// TwinCAT 3 PLC project XtsTransport
// Title: XTS Transport
// Author: D.Hauer
// ProjectVersion: 0.0.1
// Description: basic functionblocks for building XTS transport
// ProgramVersion: 3.1.4024.0
// libraries:
//   Tc2_Math, * (Beckhoff Automation GmbH)
//   Tc2_MC2, * (Beckhoff Automation GmbH)
//   Tc2_Standard, * (Beckhoff Automation GmbH)
//   Tc2_System, * (Beckhoff Automation GmbH)
//   Tc2_Utilities, * (Beckhoff Automation GmbH)
//   Tc3_McCollisionAvoidance, * (Beckhoff Automation GmbH)
//   Tc3_McCoordinatedMotion, * (Beckhoff Automation GmbH)
//   Tc3_Module, * (Beckhoff Automation GmbH)
//   Tc3_XTS_Utility, * (Beckhoff Automation GmbH)
//   VisuDialogs, * (System)
// project tree:
//   / GlobalTextList.TcGTLO, MAIN.TcPOU, PlcTask.TcTTO, PROCESS.TcPOU
//   MSG/ fb_LocalTime.TcPOU (not stored), f_MessageSet.TcPOU (not stored), GVL_MSG.TcGVL (not stored), MessageData.TcPOU (not stored), T_MESSAGE_LIST.TcVIS (not stored)
//   MSG/types/ e_Device.TcDUT (not stored), E_MessageType.TcDUT (not stored), E_MESSAGE_STATE.TcDUT (not stored), e_Subdevice.TcDUT (not stored), ST_Message.TcDUT (not stored)
//   PROCESS/ fb_Process.TcPOU, GVL_PROCESS.TcGVL, I_ExternControl_Process.TcIO, PROCESS_CONSTANTS.TcGVL
//   PROCESS/_types/ E_PROCESS_TYPE.TcDUT (not stored)
//   PROCESS/_Visualization/ PROCESS_CONTROL.TcVIS, PROCESS_XTS_TRANSPORT.TcVIS, T_GROUP_VISU.TcVIS, T_PROCESS_VISU.TcVIS, T_XPU_VISU.TcVIS
//   XTS/CaGroup/ FB_CaGroup.TcPOU, I_XtsTransport_CaGroup.TcIO (not stored)
//   XTS/CaGroup/types/ E_CA_GROUP_STATE.TcDUT (not stored), E_GROUP_CHECK.TcDUT (not stored), ST_GROUP_INFO.TcDUT
//   XTS/ GVL_XTS.TcGVL, XTS_Parameter.TcGVL
//   XTS/Mover/ fb_Mover.TcPOU, fb_MoverCtrl.TcPOU (not stored), I_XtsTransport_Mover.TcIO (not stored)
//   XTS/Mover/types/ E_MOVER_CTRL.TcDUT (not stored), E_MOVER_STATE.TcDUT (not stored), ST_GEAR_DATA.TcDUT (not stored), ST_MOVER_CTRL.TcDUT (not stored), ST_MOVER_INFO.TcDUT (not stored), ST_MOVER_STATE.TcDUT (not stored), ST_MOVE_DATA.TcDUT (not stored)
//   XTS/XtsStation/ fb_Station.TcPOU, I_XtsTransport_Station.TcIO (not stored)
//   XTS/XtsStation/_types/ E_STATION_CTRL.TcDUT (not stored), E_STATION_STATE.TcDUT (not stored), fb_Station_LinkedListCtrl.TcPOU (not stored), I_Station_LinkedList.TcIO (not stored), ST_STATION_CTRL.TcDUT (not stored), ST_STATION_LIST_RESULT.TcDUT (not stored), ST_STATION_MOVER_DATA.TcDUT (not stored), ST_STATION_PARAMETER.TcDUT (not stored), ST_STATION_STATE.TcDUT (not stored), T_NEST_OFFSET.TcDUT (not stored)
//   XTS/_types/ f_MoverIdDetectionModeToString.TcPOU, f_MoverPositionAssignementToString.TcPOU, f_XpuOperationModeToString.TcPOU (not stored), E_PROGRESS.TcDUT (not stored), f_GetProgress.TcPOU (not stored), f_GetState.TcPOU (not stored)
//   XTS/_Visualization/ GROUP_VISU.TcVIS, MOVER_VISU.TcVIS (not stored), STATION_VISU.TcVIS, Visualization Manager.TcVMO (not stored), XTS_TRANSPORT.TcVIS (not stored), XPU_VISU.TcVIS (not stored)
//   XTS/_Visualization/textlists/ TL_E_CTRL_MOVER.TcTLO (not stored), TL_E_CTRL_STATION.TcTLO (not stored), TL_E_CTRL_TRANSPORT.TcTLO (not stored), TL_E_CTRL_XPU.TcTLO (not stored)
//   XTS/Xpu/ fb_Xpu.TcPOU (not stored), fb_XpuCtrl.TcPOU (not stored)
//   XTS/Xpu/types/ E_XPU_CHECK.TcDUT (not stored), E_XPU_CTRL.TcDUT (not stored), E_XPU_INIT.TcDUT (not stored), E_XPU_STATE.TcDUT (not stored), ST_XPU_CTRL.TcDUT (not stored), ST_XPU_INFO.TcDUT (not stored), ST_XPU_STATE.TcDUT (not stored)
//   XTS/XtsTransportUnit/ fb_TransportUnit.TcPOU
//   XTS/XtsTransportUnit/types/ E_XTS_TRANSPORT_CHECK.TcDUT (not stored), E_XTS_TRANSPORT_CTRL.TcDUT (not stored), E_XTS_TRANSPORT_STATE.TcDUT (not stored), ST_XTS_TRANSPORT_CTRL.TcDUT (not stored), ST_XTS_TRANSPORT_STATE.TcDUT (not stored)

CONFIGURATION XtsTransport
    RESOURCE PLC ON TwinCAT3
        TASK PlcTask(INTERVAL := T#2ms, PRIORITY := 15);
        PROGRAM MAIN WITH PlcTask : MAIN;
        PROGRAM PROCESS WITH PlcTask : PROCESS;
    END_RESOURCE
END_CONFIGURATION

// ---- XTS/CaGroup/types/ST_GROUP_INFO.TcDUT
TYPE ST_GROUP_INFO :
STRUCT
  GroupStatusValid,
  GroupStatusBusy,
  GroupMoving, 
  GroupHoming, 
  GroupErrorStop, 
  GroupNotReady, 
  GroupStandby, 
  GroupStopping,
 
  GroupDisabled, 
  AllAxesStanding, 
  ConstantVelocity, 
  Accelerating, 
  Decelerating, 
  InPosition, 
  GroupError					  : BIT; 

  GroupErrorId					: UDINT;

  AxisCount      				: UDINT;
  AxisCountEnabled      : UDINT;

  {attribute 'displaymode':='hex'}
  CaGroupOID            : OTCID;

  CaGroupState          : E_CA_GROUP_STATE;
END_STRUCT
END_TYPE

// ---- PROCESS/GVL_PROCESS.TcGVL
{attribute 'qualified_only'}
VAR_GLOBAL

  Process           : ARRAY[1..MAX_PROCESS] OF fb_Process;  // handshake multiple XTS stations (ST_STATION_CTRL / ST_STATION_STATE)
  ItfProcess        : ARRAY[1..MAX_PROCESS] OF I_ExternControl_Process;

  StationsEnabled   : ARRAY[1..MAX_STATION] OF BOOL;        // read only; every process writes internally onto here the bits in MAIN.wEnableProcess
  MoverPerMinute    : ARRAY[1..MAX_STATION] OF UINT;
END_VAR

// ---- PROCESS/PROCESS_CONSTANTS.TcGVL
//{attribute 'qualified_only'}
VAR_GLOBAL CONSTANT
  MAX_PROCESS       : UINT := 12;

END_VAR

// ---- XTS/GVL_XTS.TcGVL
{attribute 'qualified_only'}
VAR_GLOBAL
  //---------------------------------------------------------------------------
  // XTS Station
  //  - handshakes mover in station with extern control
  //  - station parameters (positions, gap, dyn. constraints, description...)
  StationStart        : ST_STATION_PARAMETER;   // Xts transport is sending all mover to this position (CMD_TRANSPORT_START)

  // station handshaking with mover and extern process
  // station sends mover to target station/WaitPos
  // station adds mover data to LinkedList.AddTail() of target station
  Station             : ARRAY[1..MAX_STATION] OF fb_Station;
  StationList         : ARRAY[1..MAX_STATION] OF fb_Station_LinkedListCtrl;

  StationQueue        : ARRAY[1..MAX_STATION]    OF 
                        ARRAY[1..MAX_LIST_NODES] OF ST_STATION_MOVER_DATA;

  // interface for access to List methods
  StationListItf      : ARRAY[1..MAX_STATION] OF I_Station_LinkedList;

  // interface for access to station methods
  StationCtrlItf      : ARRAY[1..MAX_STATION] OF I_XtsTransport_Station;

  // ctrl / state datafields for extern control
  StationCtrl         : ARRAY[1..MAX_STATION] OF ST_STATION_CTRL;   // control for extern to write
  StationState        : ARRAY[1..MAX_STATION] OF ST_STATION_STATE;  // state for extern to read

  // station parameter
  StationParameter    : ARRAY[1..MAX_STATION] OF ST_STATION_PARAMETER;

  // static position offsets in stations
  PositionOffset      : ARRAY[1..MAX_STATION] OF T_NEST_OFFSET;


  //---------------------------------------------------------------------------
  // XTS
  // XTS TransportUnit
  //  - handles request for XPU, Group, Mover, StartUp, ReStart
  XtsTransport        : fb_TransportUnit;         // manages members of XTS transport for extern to access

  XtsTransportCtrl    : ST_XTS_TRANSPORT_CTRL;    // control of XTS transport for extern to write
  XtsTransportState   : ST_XTS_TRANSPORT_STATE;   // state   of XTS transport for extern to read


  //---------------------------------------------------------------------------
  // XPU
  // XTS-Utility checks
  Xpu             : fb_XpuCtrl;

  XpuCtrl         : ST_XPU_CTRL;
  XpuState        : ST_XPU_STATE;
  XpuInfo         : ST_XPU_INFO;
  XpuModules      : ARRAY[1..MAX_MODULE] OF Tc3_XTS_Utility.ST_InfoDataView;


  //---------------------------------------------------------------------------
  // Collision avoidance group CA
  //
  // - add mover to group
  // - build group
  // - clear group
  CaGroup         : FB_CaGroup;                   // cyclic check of CaGroup state and errors; carries methods for handling CaGroup
  CaGroupItf      : I_XtsTransport_CaGroup;       // Interface used by fb_TransportUnit

  // cyclic mapping to MOTION/Objects/CaGroup 
  CaGroupRef      : Tc3_McCoordinatedMotion.AXES_GROUP_REF;

  // Info data from CaGroup FB
  CaGroupInfo     : ST_GROUP_INFO;                // cyclic info about CaGroup for fb_TransportUnit to read
  //---------------------------------------------------------------------------

  //---------------------------------------------------------------------------
  // MC2 encapsulation, CA movement
  Mover           : ARRAY[1..MAX_MOVER] OF fb_MoverCtrl;    // MC and CA methods for mover; cyclic check for individual command on mover

  MoverCtrl       : ARRAY[1..MAX_MOVER] OF ST_MOVER_CTRL;   // control of individual mover for extern to write
  MoverState      : ARRAY[1..MAX_MOVER] OF ST_MOVER_STATE;  // state   of individual mover for extern to read

  MoverItf        : ARRAY[1..MAX_MOVER] OF I_XtsTransport_Mover;  // Interface used by fb_TransportUnit

  LastPosition    : ARRAY[1..MAX_MOVER] OF LREAL;           // on execute of any movement, value is saved here (used by fb_Mover)
  LastGap         : ARRAY[1..MAX_MOVER] OF LREAL;           // on execute of any movement, value is saved here (used by fb_Mover)

  MoverInfo       : ARRAY[1..MAX_MOVER] OF ST_MOVER_INFO;   // cyclic info about mover for extern to read

  MoveData        : ARRAY[1..MAX_MOVER] OF ST_MOVE_DATA;    // dynamic constraints for move commands
  GearData        : ARRAY[1..MAX_MOVER] OF ST_GEAR_DATA;    // dynamic constraints and positions for GearIn/GearInPosCa
  
  // cyclic mapping to MOTION/Axes
  AxisRefMover    : ARRAY[1..MAX_MOVER] OF Tc2_MC2.AXIS_REF;
  //---------------------------------------------------------------------------
END_VAR

// ---- XTS/XTS_Parameter.TcGVL
//{attribute 'qualified_only'}
VAR_GLOBAL CONSTANT
// HAUD 2024 08 09
//
//    XTS_TRANSPORT_LAYER project
//    
//    MIT License
//    
//    Copyright (c) 2024 HAUD
//    
//    Permission is hereby granted, free of charge, to any person obtaining a copy
//    of this software and associated documentation files (the "Software"), to deal
//    in the Software without restriction, including without limitation the rights
//    to use, copy, modify, merge, publish, distribute, sublicense, and/or sell
//    copies of the Software, and to permit persons to whom the Software is
//    furnished to do so, subject to the following conditions:
//    
//    The above copyright notice and this permission notice shall be included in all
//    copies or substantial portions of the Software.
//    
//    THE SOFTWARE IS PROVIDED "AS IS", WITHOUT WARRANTY OF ANY KIND, EXPRESS OR
//    IMPLIED, INCLUDING BUT NOT LIMITED TO THE WARRANTIES OF MERCHANTABILITY,
//    FITNESS FOR A PARTICULAR PURPOSE AND NONINFRINGEMENT. IN NO EVENT SHALL THE
//    AUTHORS OR COPYRIGHT HOLDERS BE LIABLE FOR ANY CLAIM, DAMAGES OR OTHER
//    LIABILITY, WHETHER IN AN ACTION OF CONTRACT, TORT OR OTHERWISE, ARISING FROM,
//    OUT OF OR IN CONNECTION WITH THE SOFTWARE OR THE USE OR OTHER DEALINGS IN THE
//    SOFTWARE.

  Version             : STRING  := '4.0.1';

  MAX_MOVER           : UINT    := TO_UINT(Tc3_XTS_Utility.TcIoXtsEnvironmentParameterList.MaxXtsMoversPerXpu);
  MAX_MODULE          : UINT    := TO_UINT(Tc3_XTS_Utility.TcIoXtsEnvironmentParameterList.MaxModulesPerPart);
  MAX_PART            : UINT    := TO_UINT(Tc3_XTS_Utility.TcIoXtsEnvironmentParameterList.MaxXtsPartsPerXpu);
  MAX_TRACK           : UINT    := TO_UINT(Tc3_XTS_Utility.TcIoXtsEnvironmentParameterList.MaxXtsTracksPerXpu);
  MAX_GROUP           : UINT    := TO_UINT(Tc3_XTS_Utility.TcIoXtsEnvironmentParameterList.MaxXtsCaGroup);

  MAX_INFO_SERVER     : UINT    := TO_UINT(Tc3_XTS_Utility.TcIoXtsEnvironmentParameterList.MaxXtsInfoServer);
  MAX_INFO_STATION    : UINT    := TO_UINT(Tc3_XTS_Utility.TcIoXtsEnvironmentParameterList.MaxXtsInfoStation);
  MAX_INFO_STOP_POS   : UINT    := TO_UINT(Tc3_XTS_Utility.TcIoXtsEnvironmentParameterList.MaxXtsStopPositionsPerStation);


  MAX_STATION         : UINT    := 28;
  MAX_STATION_NEST    : UINT    := TO_UINT(SIZEOF(ST_STATION_STATE.nMask)*8);
  // MAX_LIST_NODES      : UINT    := MAX_MOVER;
  MAX_LIST_NODES      : UINT    := 50; // visualization can not handle access to MAX_MOVER
  MAX_MASTER          : UINT    := 1;
END_VAR

// ---- PROCESS/I_ExternControl_Process.TcIO
INTERFACE I_ExternControl_Process

METHOD PUBLIC DelBitDWord : DWORD
VAR_INPUT
  inVal   : DWORD;
  bitNo   : DWORD;
END_VAR
END_METHOD

PROPERTY EnableProcess : dword
GET
END_GET
SET
END_SET
END_PROPERTY

METHOD PUBLIC GetBitDWord : BOOL
VAR_INPUT
  inVal   : DWORD;
  bitNo   : DINT;
END_VAR
END_METHOD

METHOD PUBLIC Init : BOOL
END_METHOD

PROPERTY MoverCountInQueue : uint
GET
END_GET
END_PROPERTY

PROPERTY MoverInQueue : Bool
GET
END_GET
END_PROPERTY

PROPERTY ProcessCmd : E_STATION_CTRL
SET
END_SET
END_PROPERTY

PROPERTY ProcessPerMinute : uint
GET
END_GET
END_PROPERTY

PROPERTY ProcessState : E_STATION_STATE
GET
END_GET
END_PROPERTY

PROPERTY ProcessType : e_process_type
GET
END_GET
SET
END_SET
END_PROPERTY

METHOD PUBLIC SetBitDWord : DWORD
VAR_INPUT
  inVal   : DWORD;
  bitNo   : DWORD;
END_VAR
END_METHOD

METHOD PUBLIC SetBitWord : WORD
VAR_INPUT
  inVal   : WORD;
  bitNo   : DINT;
END_VAR
END_METHOD

PROPERTY StationCount : uint
GET
END_GET
END_PROPERTY

PROPERTY StationFirst : uint
GET
END_GET
SET
END_SET
END_PROPERTY

PROPERTY TargetMask : dword
GET
END_GET
SET
END_SET
END_PROPERTY

END_INTERFACE

// ---- MAIN.TcPOU
//---------------------------------------------------------------------------------------------------------------
//
//  HAUD 2024.03.18
//
//  - XTS_TRANSPORT_LAYER
//  - transport layer members:
//    - CaGroup
//      - access to Group functions
//
//    - Mover
//      - access to MC and CA motion functions
//
//    - Xpu (ProcessingUnit)
//      - access to TcCOM Objects in Environment
//
//    - Transport Control Unit
//      - coordinates members to get XTS in defined states
//
//    - Xts Stations
//      - handshakes with extern control for mover transport
//
//  - global datafields for mrmbers in GVL_XTS namespace
//  - global interface datafields for use in members
//  - structures are assigned by reference for every member
//
//---------------------------------------------------------------------------------------------------------------
// HAUD 2024 05 29
//
//    XTS_TRANSPORT_LAYER project
//    
//    MIT License
//    
//    Copyright (c) 2024 HAUD
//    
//    Permission is hereby granted, free of charge, to any person obtaining a copy
//    of this software and associated documentation files (the "Software"), to deal
//    in the Software without restriction, including without limitation the rights
//    to use, copy, modify, merge, publish, distribute, sublicense, and/or sell
//    copies of the Software, and to permit persons to whom the Software is
//    furnished to do so, subject to the following conditions:
//    
//    The above copyright notice and this permission notice shall be included in all
//    copies or substantial portions of the Software.
//    
//    THE SOFTWARE IS PROVIDED "AS IS", WITHOUT WARRANTY OF ANY KIND, EXPRESS OR
//    IMPLIED, INCLUDING BUT NOT LIMITED TO THE WARRANTIES OF MERCHANTABILITY,
//    FITNESS FOR A PARTICULAR PURPOSE AND NONINFRINGEMENT. IN NO EVENT SHALL THE
//    AUTHORS OR COPYRIGHT HOLDERS BE LIABLE FOR ANY CLAIM, DAMAGES OR OTHER
//    LIABILITY, WHETHER IN AN ACTION OF CONTRACT, TORT OR OTHERWISE, ARISING FROM,
//    OUT OF OR IN CONNECTION WITH THE SOFTWARE OR THE USE OR OTHER DEALINGS IN THE
//    SOFTWARE.
//---------------------------------------------------------------------------------------------------------------
PROGRAM MAIN
VAR
	bInit 				: BOOL;
  eInit         : E_PROGRESS;

  nStation,
	nMover,
  nMoverSelected,
  nStationSelected,
  nStationParameter   : UINT;

  sStationText        : STRING(30);

  eTransportState     : E_XTS_TRANSPORT_STATE;
  eTransportResult    : E_PROGRESS;

  eXpuState           : E_XPU_STATE;
  eXpuResult          : E_PROGRESS;
  eXpuCheck           : E_XPU_CHECK;

  eMoverState         : E_MOVER_STATE;
  eMoverResult        : E_PROGRESS;

  sCaGroupState,
  sTransportState,
  sTransportCheck,
  sTransportResult,
  sXpuState,
  sXpuResult,
  sXpuCheck,
  sXpuOpMode,
  sXpuMoverdetectionMode,
  sXpuMoverAssignement,
  sMoverState,
  sMoverResult,
  sStationState,
  sStationStateMask,
  sStationCtrlMask        : STRING;

  bStationEnable,
  bStationEnter,
  bStationStart,
  bStationDone,
  bStationOut,
  bStationGone            : BOOL;

  tStationSelectedQueue   : ARRAY[1..MAX_LIST_NODES] OF ST_STATION_MOVER_DATA;

  tonWriteLog             : Tc2_Standard.TON;
  tWriteLog               : TIME := T#5S;
END_VAR

//############################################################################
// Local time; used for timestamps
//############################################################################
GVL_MSG.fbLocalTime(
                    sLocalTime                => GVL_MSG.sLocalTime, 
                    dtLocalTime               => GVL_MSG.dtLocalTime);
//############################################################################

//############################################################################
// 	example for init sequence
//############################################################################	
IF NOT bInit
THEN
  CASE eInit
  OF
    E_PROGRESS.PROGRESS_INVALID,
    E_PROGRESS.PROGRESS_DONE:         // clear command interface
      eInit                                   := E_PROGRESS.PROGRESS_BUSY;
      GVL_XTS.XpuCtrl.Cmd                     := E_XPU_CTRL.XTS_CMD_NULL;
      GVL_MSG.MessageLevelXpu                 := GVL_MSG.MessageLevel;
      FOR nStation := 1 TO MAX_STATION
      DO
        GVL_MSG.MessageLevelStations[nStation]:= GVL_MSG.MessageLevel;
      END_FOR
      FOR nMover := 1 TO MAX_MOVER
      DO
        GVL_MSG.MessageLevelMovers[nMover]    := GVL_MSG.MessageLevel;
      END_FOR


    E_PROGRESS.PROGRESS_BUSY:         // init Xpu, ProcessingUnit, MotorModules
      eInit                                   := E_PROGRESS.PROGRESS_PREPARE;
      GVL_XTS.XpuCtrl.Cmd                     := E_XPU_CTRL.XTS_CMD_INIT;

    E_PROGRESS.PROGRESS_PREPARE:      // wait for init to be done
      IF (GVL_XTS.XpuState.State      = E_XPU_STATE.XTS_INIT + E_PROGRESS.PROGRESS_DONE)
      THEN
        eInit                                 := E_PROGRESS.PROGRESS_STARTUP;
        GVL_XTS.XpuCtrl.Cmd                   := E_XPU_CTRL.XTS_IDLE;
      END_IF

    E_PROGRESS.PROGRESS_STARTUP:      // assign mover interfaces
      eInit                                   := E_PROGRESS.PROGRESS_CHECK;
      FOR nMover := 1 TO MAX_MOVER
      DO
        GVL_XTS.MoverItf[nMover]              := GVL_XTS.Mover[nMover];
      END_FOR

    E_PROGRESS.PROGRESS_CHECK:        // assign CaGroup interface
      eInit                                   := E_PROGRESS.PROGRESS_OCCUPIED;
      GVL_XTS.CaGroupItf                      := GVL_XTS.CaGroup;

    E_PROGRESS.PROGRESS_OCCUPIED:     // StartStation for XtsTransportCtrl.Cmd := E_XTS_TRANSPORT_CTRL.CMD_TRANSPORT_START;
      eInit                                   := E_PROGRESS.PROGRESS_WORKING;
      // where to start?
      GVL_XTS.XtsTransport.StartStationIndex  := 28;

      // Start Position parameters
      GVL_XTS.StationStart.rPosWait           := GVL_XTS.StationParameter[28].rPosWait;
      GVL_XTS.StationStart.rGap               :=    100.0;
      GVL_XTS.StationStart.rVelo              :=   1250.0;
      GVL_XTS.StationStart.rAccDec            :=  12000.0;
      GVL_XTS.StationStart.rJerk              := 400000.0;

    E_PROGRESS.PROGRESS_WORKING:
      bInit                                           := TRUE;
      eInit                                           := E_PROGRESS.PROGRESS_DONE;
  END_CASE
END_IF

//############################################################################
// 	XTS Transport Unit
//############################################################################
//  - main control function block for transport layer
//  - requires access to member controls
//    - Xpu
//    - CaGroup
//    - Mover
//    - Station Control
//    - Station LinkedList Interface
//############################################################################
//
// cyclic call
GVL_XTS.XtsTransport();

// main control
GVL_XTS.XtsTransport.Ctrl               REF= GVL_XTS.XtsTransportCtrl;   // main control
GVL_XTS.XtsTransport.State              REF= GVL_XTS.XtsTransportState;  // main state
                                        
// member controls                      
GVL_XTS.XtsTransport.XpuCtrl            REF= GVL_XTS.XpuCtrl;
GVL_XTS.XtsTransport.XpuState           REF= GVL_XTS.XpuState;
GVL_XTS.XtsTransport.XpuInfo            REF= GVL_XTS.XpuInfo;
                                        
GVL_XTS.XtsTransport.GroupItf           :=   GVL_XTS.CaGroupItf;
GVL_XTS.XtsTransport.GroupInfo          REF= GVL_XTS.CaGroupInfo;
                                        
GVL_XTS.XtsTransport.MoverItf           REF= GVL_XTS.MoverItf;
GVL_XTS.XtsTransport.MoverInfo          REF= GVL_XTS.MoverInfo;
                                        
GVL_XTS.XtsTransport.StationStart       REF= GVL_XTS.StationStart;      // start position for E_XTS_TRANSPORT_CTRL.CMD_TRANSPORT_START
GVL_XTS.XtsTransport.StationCtrlItf     REF= GVL_XTS.StationCtrlItf;    // station interfaces are required for accessing station methods
GVL_XTS.XtsTransport.StationListsItf    REF= GVL_XTS.StationListItf;    // list interface is required for access to linked list methods
//############################################################################



//############################################################################
// 	XTS Stations
//############################################################################	
FOR nStation := 1 TO MAX_STATION
DO
  GVL_XTS.Station[nStation].StationId   := nStation;
  GVL_XTS.Station[nStation].MessageLevel:= GVL_MSG.MessageLevelStations[nStation];

  GVL_XTS.StationListItf[nStation]      := GVL_XTS.StationList[nStation];   // interfaces for list methods
  GVL_XTS.StationCtrlItf[nStation]      := GVL_XTS.Station[nStation];       // interfaces for station methods

  GVL_XTS.Station[nStation].Ctrl        REF= GVL_XTS.StationCtrl;           // station ctrl from extern
  GVL_XTS.Station[nStation].State       REF= GVL_XTS.StationState;          // station state to extern

  GVL_XTS.Station[nStation].ItfStations REF= GVL_XTS.StationListItf;        // give every station all list interfaces for writing mover tickets
  GVL_XTS.Station[nStation].ItfMover    REF= GVL_XTS.MoverItf;              // give every station all mover interfaces for movement in / out of station
  GVL_XTS.Station[nStation].Mover       REF= GVL_XTS.AxisRefMover;          // AXIS_REF to read infos from
  GVL_XTS.Station[nStation].MoverOffset REF= GVL_XTS.PositionOffset;        // static offsets for all stations, all movers, all stop positions


  GVL_XTS.Station[nStation].StationParameter  REF= GVL_XTS.StationParameter;// give every station all station parameters for sending to WaitPos of target station

  // cyclic call
  GVL_XTS.Station[nStation].Cycle();                                        // cycle for handshaking with extern

  // Queue data for each station
  GVL_XTS.StationQueue[nStation]        := GVL_XTS.StationListItf[nStation].Data;
END_FOR
//############################################################################



//############################################################################
// 	XPU environment
//############################################################################	
GVL_XTS.Xpu.XpuInstance               :=   1;
GVL_XTS.Xpu.MessageLevel              :=   GVL_MSG.MessageLevelXpu;

GVL_XTS.Xpu.Ctrl                      REF= GVL_XTS.XpuCtrl;
GVL_XTS.Xpu.State                     REF= GVL_XTS.XpuState;
GVL_XTS.Xpu.XpuModuleInfoData         REF= GVL_XTS.XpuModules;

GVL_XTS.Xpu.CaGroupOID                :=   GVL_XTS.CaGroup.GroupInfo.CaGroupOID;

// cyclic call
GVL_XTS.Xpu();
GVL_XTS.XpuInfo                       :=   GVL_XTS.Xpu.XpuInfo;
//############################################################################


//############################################################################	
// 	CA-Group Class
//############################################################################	
// assignment
GVL_XTS.CaGroup.AxisRef               REF= GVL_XTS.AxisRefMover;
GVL_XTS.CaGroup.GroupRef              REF= GVL_XTS.CaGroupRef;

GVL_XTS.CaGroup.MessageLevel          :=   GVL_MSG.MessageLevel;

// cyclic call
GVL_XTS.CaGroup.InfoCycle(TRUE); // read group status

// InfoData from group
GVL_XTS.CaGroupInfo                   :=   GVL_XTS.CaGroup.GroupInfo;

// Interface of CaGroup
GVL_XTS.CaGroupItf                    :=   GVL_XTS.CaGroup;
//############################################################################


//############################################################################
// Mover Class	
//############################################################################	
FOR nMover := 1 TO MAX_MOVER
DO
  GVL_XTS.Mover[nMover].MoverId       :=   nMover;
  GVL_XTS.Mover[nMover].RailLength    :=   GVL_XTS.Xpu.RailLength;  // mover needs RailLength, in order to calc absolute position from modulo input
  GVL_XTS.Mover[nMover].MessageLevel  :=   GVL_MSG.MessageLevelMovers[nMover];

  GVL_XTS.Mover[nMover].Ctrl          REF= GVL_XTS.MoverCtrl;       // mover control from extern
  GVL_XTS.Mover[nMover].State         REF= GVL_XTS.MoverState;      // mover state to extern

  GVL_XTS.Mover[nMover].MoveData      REF= GVL_XTS.MoveData;        // dyn constraints for extern to write
  GVL_XTS.Mover[nMover].GearData      REF= GVL_XTS.GearData;        // GearIn/GearInPosCa data fro extern to write

  // assignment	
  GVL_XTS.Mover[nMover].Mover         REF= GVL_XTS.AxisRefMover[nMover];  // axis reference to Mover function block
  GVL_XTS.Mover[nMover].LastGap       REF= GVL_XTS.LastGap[nMover];       // reference to last used gap value datafield
  GVL_XTS.Mover[nMover].LastPosition  REF= GVL_XTS.LastPosition[nMover];  // reference to last position datafield

  GVL_XTS.Mover[nMover].MoverInfo		  REF= GVL_XTS.MoverInfo[nMover];     // refernence to mover info data (ActPos, SetPos, ...)

  GVL_XTS.MoverItf[nMover]            :=   GVL_XTS.Mover[nMover];

  // cyclic call
  GVL_XTS.Mover[nMover].Cycle();  // call AXIS_REF()
  GVL_XTS.Mover[nMover]();        // call Ctrl/State
END_FOR


//############################################################################


//############################################################################
// /logging
//############################################################################
tonWriteLog(IN:= TRUE, PT := tWriteLog);

IF (tonWriteLog.Q)
THEN
  MessageData.bWriteFile      := TRUE;
  tonWriteLog(IN:= FALSE);
END_IF

//-----------------------------------------------------------------------------------------------------------------
// write message list to file
//-----------------------------------------------------------------------------------------------------------------
MessageData(pList			        := ADR(GVL_MSG.Messages),
			      pLocalTime        := ADR(GVL_MSG.dtLocalTime), 
			      bBusy=> );

// clear write trigger
IF MessageData.bWriteFile AND
   MessageData.bDone
THEN
  MessageData.bWriteFile      := FALSE;
END_IF
//############################################################################
// logging/
//############################################################################



//############################################################################
// Visualization data	
//############################################################################	
// get enumerations from XPU for visu:
eTransportState                       := f_GetState   (GVL_XTS.XtsTransportState.State);
eTransportResult                      := f_GetProgress(GVL_XTS.XtsTransportState.State);

eXpuState                             := f_GetState   (GVL_XTS.XpuState.State);
eXpuResult                            := f_GetProgress(GVL_XTS.XpuState.State);

eXpuCheck                             := GVL_XTS.XpuState.Check;

// display xpu state and result in visu
// get strings and info
sCaGroupState                         := TO_STRING(GVL_XTS.CaGroupInfo.CaGroupState);

sTransportState                       := TO_STRING(eTransportState);
sTransportCheck                       := TO_STRING(GVL_XTS.XtsTransportState.Check);
sTransportResult                      := TO_STRING(eTransportResult);

sXpuState                             := TO_STRING(eXpuState);
sXpuResult                            := TO_STRING(eXpuResult);
sXpuCheck                             := TO_STRING(eXpuCheck);

sXpuOpMode                            := GVL_XTS.Xpu.OpModeToString();
sXpuMoverdetectionMode                := GVL_XTS.Xpu.IdDetectionModeToString();
sXpuMoverAssignement                  := GVL_XTS.Xpu.MoverPositionAssignementToString();

nMoverSelected                        := SEL((nMoverSelected<1), nMoverSelected, 1);
nMoverSelected                        := SEL((nMoverSelected>MAX_MOVER), nMoverSelected, MAX_MOVER);

nStationSelected                      := SEL((nStationSelected<1), nStationSelected, 1);
nStationSelected                      := SEL((nStationSelected>MAX_STATION), nStationSelected, MAX_STATION);

bStationEnable                        := SEL((GVL_XTS.StationCtrl[nStationSelected].eCmd = E_STATION_CTRL.STATION_ENABLE),        FALSE, TRUE);
bStationEnter                         := SEL((GVL_XTS.StationCtrl[nStationSelected].eCmd = E_STATION_CTRL.STATION_MOVER_ENTER),   FALSE, TRUE);
bStationStart                         := SEL((GVL_XTS.StationCtrl[nStationSelected].eCmd = E_STATION_CTRL.STATION_PROCESS_START), FALSE, TRUE);
bStationDone                          := SEL((GVL_XTS.StationCtrl[nStationSelected].eCmd = E_STATION_CTRL.STATION_PROCESS_DONE),  FALSE, TRUE);
bStationOut                           := SEL((GVL_XTS.StationCtrl[nStationSelected].eCmd = E_STATION_CTRL.STATION_MOVER_OUT),     FALSE, TRUE);
bStationGone                          := SEL((GVL_XTS.StationCtrl[nStationSelected].eCmd = E_STATION_CTRL.STATION_MOVER_GONE),    FALSE, TRUE);

eMoverState                           := f_GetState   (GVL_XTS.MoverState[nMoverSelected].State);
eMoverResult                          := f_GetProgress(GVL_XTS.MoverState[nMoverSelected].State);

sMoverState                           := TO_STRING(eMoverState);
sMoverResult                          := TO_STRING(eMoverResult);

sStationState                         := TO_STRING(GVL_XTS.StationState[nStationSelected].eState);
sStationStateMask                     := Tc2_Utilities.BYTE_TO_BINSTR(GVL_XTS.StationState[nStationSelected].nMask, 8);
sStationCtrlMask                      := Tc2_Utilities.BYTE_TO_BINSTR(GVL_XTS.StationCtrl[nStationSelected].nMask, 8);

tStationSelectedQueue                 := GVL_XTS.StationQueue[nStationSelected];

END_PROGRAM

// ---- PROCESS.TcPOU
//---------------------------------------------------------------------------------------------------------------
//
//  HAUD 2024.04.13
//
//  - ExternControl for XtsTransport
//
//  - example project for controlling XTS transport layer
//  - transport layer members:
//
//      HAUD 2024 04 30 - introduction of fb_UnitControl as interface to APPLICATION
//
//    - fb_UnitControl
//      - groups commands into sequences for APPLICATION
//      - handles XtsTransport
//      - handles fb_Process
//
//    - fb_Process
//      - groups XtsStations for processes
//      - synced handshakes with all assigned XtsStations
//
//    - Transport Control Unit
//      - mapped from XtsTransport GVL_XTS.TransportCtrl / GVL_XTS.TransportState
//        - Info for CaGroup
//        - Info for Xpu
//
//      - coordinates members to get XTS in defined states
//
//    - Xts Stations
//      - handshakes for mover transport
//
//---------------------------------------------------------------------------------------------------------------
// This SOFTWARE is provided as an Exemple by THE PROVIDER "as is" and "with all faults." THE PROVIDER makes no 
// representations or warranties of any kind concerning the safety, suitability, lack of viruses, inaccuracies, 
// typographical errors, or other harmful components of this SOFTWARE. There are inherent dangers in the use of 
// any software, and you are solely responsible for determining whether this SOFTWARE is compatible with your 
// equipment and other software installed on your equipment. You are also solely responsible for the protection 
// of your equipment and backup of your data, and THE PROVIDER will not be liable for any damages you may suffer 
// in connection with using, modifying, or distributing this SOFTWARE.
//---------------------------------------------------------------------------------------------------------------
PROGRAM PROCESS
VAR
  bInit,
  bStart              : BOOL;       // start bit for AUTO
  eInit               : E_PROGRESS; // process initialization

  eTransportCmd,
  eTransportCmdOld    : E_XTS_TRANSPORT_CTRL; // ctrl input sequence

  eTransportState,
  eTransportStateOld  : E_XTS_TRANSPORT_STATE;// state output sequence

  eTransportResult,
  eStateStart         : E_PROGRESS;

  nProcess,
  nStation            : UINT;

  tProcess            : ARRAY[1..MAX_PROCESS] OF TIME;
  tonProcess          : ARRAY[1..MAX_PROCESS] OF Tc2_Standard.TON;

  {attribute 'displaymode':='bin'}
  wEnableProcess      : ARRAY[1..MAX_PROCESS] OF DWORD;  // switch XTS stations on/off here (one word per process --> max. 16 stations each)

  {attribute 'displaymode':='bin'}
  wInitProcess        : WORD;  // processes init

//  eProcessCmd         : ARRAY[1..MAX_PROCESS] OF E_STATION_CTRL;
//  eProcessState       : ARRAY[1..MAX_PROCESS] OF E_STATION_STATE;

  // visualization vars
  nMoverSelected,
  nStationSelected,
  nProcessSelected,
  nStationParameter,
  nProcessParameter   : UINT;

  eXpuState           : E_XPU_STATE;
  eXpuResult          : E_PROGRESS;
  eXpuCheck           : E_XPU_CHECK;

  eMoverState         : E_MOVER_STATE;
  eMoverResult        : E_PROGRESS;

  sCaGroupState,
  sTransportState,
  sTransportCheck,
  sTransportResult,
  sXpuState,
  sXpuResult,
  sXpuCheck,
  sXpuOpMode,
  sXpuMoverdetectionMode,
  sXpuMoverAssignement,
  sMoverState,
  sMoverResult,
  sStationState,
  sStationStateMask,
  sStationCtrlMask,
  sProcessEnableMask        : STRING;

  bStationEnable,
  bStationEnter,
  bStationStart,
  bStationDone,
  bStationOut,
  bStationGone            : BOOL;

  sStationText            : STRING;
END_VAR

//#############################################################################
// Visualization data	
//#############################################################################	
VisuData();
//
//#############################################################################
// check for changed Cmd on XtsTransportCtrl.Cmd
//#############################################################################
//
eTransportCmd                         := GVL_XTS.XtsTransportCtrl.Cmd;
//
IF (eTransportCmd <> eTransportCmdOld)
THEN
  eTransportCmdOld                    := eTransportCmd;
  bStart                              := FALSE;
  bEmptySerialStation                 := FALSE;
  eStateStart                         := E_PROGRESS.PROGRESS_INIT;
  memset(ADR(wEnableProcess), 0, SIZEOF(wEnableProcess));

  CASE eTransportCmd
  OF
    E_XTS_TRANSPORT_CTRL.CMD_INIT:
      bInit                           := FALSE;

  ELSE
    IF bInit
    THEN
      CASE eTransportCmd
      OF
        E_XTS_TRANSPORT_CTRL.CMD_IDLE,
        E_XTS_TRANSPORT_CTRL.CMD_TRANSPORT_START:
          FOR nProcess := 1 TO MAX_PROCESS
          DO
            ;//eProcessCmd[nProcess]     := E_STATION_CTRL.STATION_DISABLE;
          END_FOR
      END_CASE
    END_IF
  END_CASE
END_IF
//
//
//#############################################################################
// check for changed state on XtsTransportState.State
//#############################################################################
//
IF (GVL_XTS.XtsTransportState.State <> eTransportStateOld)
THEN
  CASE (GVL_XTS.XtsTransportState.State MOD E_PROGRESS.PROGRESS_DONE)
  OF
    E_XTS_TRANSPORT_STATE.TRANSPORT_START:
      CASE eStateStart
      OF
        E_PROGRESS.PROGRESS_INIT:
          IF GVL_XTS.XtsTransportState.GroupInfo.AllAxesStanding
          THEN
            eStateStart               := E_PROGRESS.PROGRESS_BUSY;
            memset(ADR(wEnableProcess), 0, SIZEOF(wEnableProcess));
          END_IF

        E_PROGRESS.PROGRESS_BUSY:
          eStateStart                   := E_PROGRESS.PROGRESS_PREPARE;
          FOR nProcess := 1 TO MAX_PROCESS
          DO
            FOR nStation := 1 TO GVL_PROCESS.Process[nProcess].StationCount
            DO
              wEnableProcess[nProcess]  := GVL_PROCESS.Process[nProcess].SetBitDWord(wEnableProcess[nProcess],(nStation-1));
            END_FOR
            GVL_PROCESS.Process[nProcess].EnableProcess := TO_WORD(wEnableProcess[nProcess]);
          END_FOR

        E_PROGRESS.PROGRESS_PREPARE:
          eStateStart                   := E_PROGRESS.PROGRESS_STARTUP;
          FOR nProcess := 1 TO MAX_PROCESS
          DO
            IF (nProcess = MAX_PROCESS)
            THEN
              GVL_PROCESS.Process[nProcess].TargetMask := wEnableProcess[1];
            ELSE
              GVL_PROCESS.Process[nProcess].TargetMask := wEnableProcess[nProcess+1];
            END_IF
          END_FOR

        E_PROGRESS.PROGRESS_STARTUP:
          eStateStart                   := E_PROGRESS.PROGRESS_CHECK;

        E_PROGRESS.PROGRESS_CHECK:
          eStateStart                 := E_PROGRESS.PROGRESS_OCCUPIED;
          FOR nProcess := 1 TO MAX_PROCESS
          DO
            IF NOT (GVL_PROCESS.Process[nProcess].EnableProcess = wEnableProcess[nProcess])
            THEN
              eStateStart             := E_PROGRESS.PROGRESS_CHECK;
            END_IF
          END_FOR

        E_PROGRESS.PROGRESS_OCCUPIED:
          eTransportStateOld          := GVL_XTS.XtsTransportState.State;
          bStart                      := TRUE;
      END_CASE

  ELSE
    eTransportStateOld                := GVL_XTS.XtsTransportState.State;

    CASE (GVL_XTS.XtsTransportState.State MOD E_PROGRESS.PROGRESS_ERROR)
    OF
      E_XTS_TRANSPORT_STATE.TRANSPORT_START:
        bStart                        := FALSE;

    END_CASE
  END_CASE
END_IF
//
//#############################################################################
//#############################################################################
//
IF NOT bInit
THEN
  Init();
END_IF
//#############################################################################
//#############################################################################
// cyclic call to processes
//#############################################################################
FOR nProcess := 1 TO MAX_PROCESS
DO
  GVL_PROCESS.Process[nProcess].Cycle();

  GVL_PROCESS.Process[nProcess].EnabledStation    := ADR(GVL_PROCESS.StationsEnabled);  // enabled process: for other processes to read
  GVL_PROCESS.Process[nProcess].MoverPerMinute    := ADR(GVL_PROCESS.MoverPerMinute);

  GVL_PROCESS.Process[nProcess].StationCtrl       := ADR(GVL_XTS.StationCtrl);
  GVL_PROCESS.Process[nProcess].StationState      := ADR(GVL_XTS.StationState);

  GVL_PROCESS.ItfProcess[nProcess]                := GVL_PROCESS.Process[nProcess]; 
END_FOR


//#############################################################################
// process workers
//#############################################################################


//#############################################################################
//
IF NOT (bInit) THEN RETURN; END_IF
//
//#############################################################################
//#############################################################################

AUTO();












//#############################################################################

ACTION AUTO:


IF NOT bStart THEN RETURN; END_IF


FOR nProcess := 1 TO MAX_PROCESS
DO
  CASE GVL_PROCESS.ItfProcess[nProcess].ProcessState
  OF
    E_STATION_STATE.STATION_DISABLE:
      GVL_PROCESS.ItfProcess[nProcess].ProcessCmd       := E_STATION_CTRL.STATION_ENABLE;

    E_STATION_STATE.STATION_MOVER_ENTER:
      CASE GVL_PROCESS.ItfProcess[nProcess].ProcessType
      OF
        E_PROCESS_TYPE.DISTRIBUTOR:
          GVL_PROCESS.ItfProcess[nProcess].ProcessCmd := E_STATION_CTRL.STATION_MOVER_SEND;
(*
          IF (GVL_XTS.StationState[GVL_PROCESS.ItfProcess[nProcess].StationFirst].rMoverModPos > GVL_XTS.StationParameter[GVL_PROCESS.ItfProcess[nProcess].StationFirst].rPosWait-5.0)// AND
          THEN
            GVL_PROCESS.ItfProcess[nProcess].ProcessCmd := E_STATION_CTRL.STATION_MOVER_SEND;
          END_IF
*)
      ELSE
          GVL_PROCESS.ItfProcess[nProcess].ProcessCmd   := E_STATION_CTRL.STATION_MOVER_ENTER;
      END_CASE

    E_STATION_STATE.STATION_PROCESS_START:
      tonProcess[nProcess](IN:= FALSE, PT:= tProcess[nProcess]);
      GVL_PROCESS.ItfProcess[nProcess].ProcessCmd       := E_STATION_CTRL.STATION_PROCESS_START;

    E_STATION_STATE.STATION_PROCESS_DONE:
      tonProcess[nProcess](IN:= TRUE, PT:= tProcess[nProcess]);
      IF tonProcess[nProcess].Q
      THEN
        GVL_PROCESS.ItfProcess[nProcess].ProcessCmd     := E_STATION_CTRL.STATION_PROCESS_DONE;
      END_IF

    E_STATION_STATE.STATION_MOVER_OUT:
      GVL_PROCESS.ItfProcess[nProcess].ProcessCmd       := E_STATION_CTRL.STATION_MOVER_OUT;

  END_CASE
END_FOR
END_ACTION

METHOD Init
VAR_INPUT
END_VAR
CASE eInit
OF
  E_PROGRESS.PROGRESS_INVALID,
  E_PROGRESS.PROGRESS_DONE:
    StationParameterInit();
    ProcessParameterInit();

    bStart                          := FALSE;
    eInit                           := E_PROGRESS.PROGRESS_INIT;
    GVL_XTS.XtsTransportCtrl.Cmd    := E_XTS_TRANSPORT_CTRL.CMD_NULL;

  E_PROGRESS.PROGRESS_INIT:
    IF (GVL_XTS.XtsTransportState.XpuInfo.IdDetectionValid) OR
       (GVL_XTS.XtsTransportState.XpuInfo.OperationMode = 1) // Simulation
    THEN
      GVL_XTS.XtsTransportCtrl.Cmd  := E_XTS_TRANSPORT_CTRL.CMD_INIT;

      IF (GVL_xts.XtsTransportState.State = E_XTS_TRANSPORT_STATE.TRANSPORT_INIT + E_PROGRESS.PROGRESS_DONE)
      THEN
        GVL_XTS.XtsTransportCtrl.Cmd:= E_XTS_TRANSPORT_CTRL.CMD_IDLE;
        eInit                       := E_PROGRESS.PROGRESS_BUSY;
      END_IF
    END_IF

  E_PROGRESS.PROGRESS_BUSY:
    eInit                           := E_PROGRESS.PROGRESS_PREPARE;
    wInitProcess                    := 0;

  E_PROGRESS.PROGRESS_PREPARE:

    FOR nProcess := 1 TO MAX_PROCESS
    DO
      GVL_PROCESS.Process[nProcess].TargetMask        := 0;
      GVL_PROCESS.Process[nProcess].ProcessCmd        := E_STATION_CTRL.STATION_INIT;
      IF (GVL_PROCESS.Process[nProcess].ProcessState = E_STATION_STATE.STATION_INIT)
      THEN
        wInitProcess                := GVL_PROCESS.Process[nProcess].SetBitWord(wInitProcess,  (nProcess-1));
      END_IF
    END_FOR
    IF (wInitProcess = EXPT(2,MAX_PROCESS)-1)
    THEN
      eInit                         := E_PROGRESS.PROGRESS_STARTUP;
    END_IF

  E_PROGRESS.PROGRESS_STARTUP:
    FOR nProcess := 1 TO MAX_PROCESS
    DO
      GVL_PROCESS.Process[nProcess].ProcessCmd         := E_STATION_CTRL.STATION_DISABLE;
    END_FOR
    bInit                           := TRUE;
    eInit                           := E_PROGRESS.PROGRESS_DONE;
END_CASE
END_METHOD

ACTION ProcessParameterInit:


// Beladen
//---------------------------------------------------------------------------------------
//---------------------------------------------------------------------------------------
  nProcessParameter   := 1;
  tProcess[nProcessParameter]             := T#3000MS;
  GVL_PROCESS.Process[nProcessParameter].ProcessType   := E_PROCESS_TYPE.PARALLEL_STRICT;
  GVL_PROCESS.Process[nProcessParameter].StationFirst  :=  1;
  GVL_PROCESS.Process[nProcessParameter].StationLast   :=  5;
  GVL_PROCESS.Process[nProcessParameter].TargetFirst   :=  6;
  GVL_PROCESS.Process[nProcessParameter].TargetLast    := 10;

// WKZ_1
//---------------------------------------------------------------------------------------
//---------------------------------------------------------------------------------------
  nProcessParameter   := 2;
  tProcess[nProcessParameter]             := T#3000MS;
  GVL_PROCESS.Process[nProcessParameter].ProcessType   := E_PROCESS_TYPE.PARALLEL_STRICT;
  GVL_PROCESS.Process[nProcessParameter].StationFirst  :=  6;
  GVL_PROCESS.Process[nProcessParameter].StationLast   := 10;
  GVL_PROCESS.Process[nProcessParameter].TargetFirst   := 11;
  GVL_PROCESS.Process[nProcessParameter].TargetLast    := 11;

// DISTRIBUTOR_SCAN
//---------------------------------------------------------------------------------------
//---------------------------------------------------------------------------------------
  nProcessParameter   := 3;
  tProcess[nProcessParameter]             := T#0MS;
  GVL_PROCESS.Process[nProcessParameter].ProcessType   := E_PROCESS_TYPE.DISTRIBUTOR;
  GVL_PROCESS.Process[nProcessParameter].StationFirst  := 11;
  GVL_PROCESS.Process[nProcessParameter].StationLast   := 11;
  GVL_PROCESS.Process[nProcessParameter].TargetFirst   := 12;
  GVL_PROCESS.Process[nProcessParameter].TargetLast    := 13;

// SCANNER
//---------------------------------------------------------------------------------------
//---------------------------------------------------------------------------------------
  nProcessParameter   := 4;
  tProcess[nProcessParameter]             := T#1000MS;
  GVL_PROCESS.Process[nProcessParameter].ProcessType   := E_PROCESS_TYPE.PARALLEL_STRICT;
  GVL_PROCESS.Process[nProcessParameter].StationFirst  := 12;
  GVL_PROCESS.Process[nProcessParameter].StationLast   := 13;
  GVL_PROCESS.Process[nProcessParameter].TargetFirst   := 14;
  GVL_PROCESS.Process[nProcessParameter].TargetLast    := 14;

// DISTRIBUTOR_WKZ_2
//---------------------------------------------------------------------------------------
//---------------------------------------------------------------------------------------
  nProcessParameter   := 5;
  tProcess[nProcessParameter]             := T#0MS;
  GVL_PROCESS.Process[nProcessParameter].ProcessType   := E_PROCESS_TYPE.DISTRIBUTOR;
  GVL_PROCESS.Process[nProcessParameter].StationFirst  := 14;
  GVL_PROCESS.Process[nProcessParameter].StationLast   := 14;
  GVL_PROCESS.Process[nProcessParameter].TargetFirst   := 15;
  GVL_PROCESS.Process[nProcessParameter].TargetLast    := 19;

// WKZ_2
//---------------------------------------------------------------------------------------
//---------------------------------------------------------------------------------------
  nProcessParameter   := 6;
  tProcess[nProcessParameter]             := T#3000MS;
  GVL_PROCESS.Process[nProcessParameter].ProcessType   := E_PROCESS_TYPE.PARALLEL_STRICT;
  GVL_PROCESS.Process[nProcessParameter].StationFirst  := 15;
  GVL_PROCESS.Process[nProcessParameter].StationLast   := 19;
  GVL_PROCESS.Process[nProcessParameter].TargetFirst   := 20;
  GVL_PROCESS.Process[nProcessParameter].TargetLast    := 20;

// CAMERA_ADJUST
//---------------------------------------------------------------------------------------
//---------------------------------------------------------------------------------------
  nProcessParameter   := 7;
  tProcess[nProcessParameter]             := T#400MS;
  GVL_PROCESS.Process[nProcessParameter].ProcessType   := E_PROCESS_TYPE.SINGLE;
  GVL_PROCESS.Process[nProcessParameter].StationFirst  := 20;
  GVL_PROCESS.Process[nProcessParameter].StationLast   := 20;
  GVL_PROCESS.Process[nProcessParameter].TargetFirst   := 21;
  GVL_PROCESS.Process[nProcessParameter].TargetLast    := 21;

// DISTRIBUTOR_CAMERA
//---------------------------------------------------------------------------------------
//---------------------------------------------------------------------------------------
  nProcessParameter   := 8;
  tProcess[nProcessParameter]             := T#0MS;
  GVL_PROCESS.Process[nProcessParameter].ProcessType   := E_PROCESS_TYPE.DISTRIBUTOR;
  GVL_PROCESS.Process[nProcessParameter].StationFirst  := 21;
  GVL_PROCESS.Process[nProcessParameter].StationLast   := 21;
  GVL_PROCESS.Process[nProcessParameter].TargetFirst   := 22;
  GVL_PROCESS.Process[nProcessParameter].TargetLast    := 24;

// CAMERA
//---------------------------------------------------------------------------------------
//---------------------------------------------------------------------------------------
  nProcessParameter   := 9;
  tProcess[nProcessParameter]             := T#1000MS;
  GVL_PROCESS.Process[nProcessParameter].ProcessType   := E_PROCESS_TYPE.PARALLEL_STRICT;
  GVL_PROCESS.Process[nProcessParameter].StationFirst  := 22;
  GVL_PROCESS.Process[nProcessParameter].StationLast   := 24;
  GVL_PROCESS.Process[nProcessParameter].TargetFirst   := 25;
  GVL_PROCESS.Process[nProcessParameter].TargetLast    := 25;

// DISTRIBUTOR_UNLOAD
//---------------------------------------------------------------------------------------
//---------------------------------------------------------------------------------------
  nProcessParameter   := 10;
  tProcess[nProcessParameter]             := T#0MS;
  GVL_PROCESS.Process[nProcessParameter].ProcessType   := E_PROCESS_TYPE.DISTRIBUTOR;
  GVL_PROCESS.Process[nProcessParameter].StationFirst  := 25;
  GVL_PROCESS.Process[nProcessParameter].StationLast   := 25;
  GVL_PROCESS.Process[nProcessParameter].TargetFirst   := 26;
  GVL_PROCESS.Process[nProcessParameter].TargetLast    := 27;

// UNLOAD
//---------------------------------------------------------------------------------------
//---------------------------------------------------------------------------------------
  nProcessParameter   := 11;
  tProcess[nProcessParameter]             := T#1050MS;
  GVL_PROCESS.Process[nProcessParameter].ProcessType   := E_PROCESS_TYPE.PARALLEL_STRICT;
  GVL_PROCESS.Process[nProcessParameter].StationFirst  := 26;
  GVL_PROCESS.Process[nProcessParameter].StationLast   := 27;
  GVL_PROCESS.Process[nProcessParameter].TargetFirst   := 28;
  GVL_PROCESS.Process[nProcessParameter].TargetLast    := 28;

// DISTRIBUTOR_LOAD
//---------------------------------------------------------------------------------------
//---------------------------------------------------------------------------------------
  nProcessParameter   := 12;
  tProcess[nProcessParameter]             := T#0MS;
  GVL_PROCESS.Process[nProcessParameter].ProcessType   := E_PROCESS_TYPE.DISTRIBUTOR;
  GVL_PROCESS.Process[nProcessParameter].StationFirst  := 28;
  GVL_PROCESS.Process[nProcessParameter].StationLast   := 28;
  GVL_PROCESS.Process[nProcessParameter].TargetFirst   := 1;
  GVL_PROCESS.Process[nProcessParameter].TargetLast    := 5;
END_ACTION

ACTION StationParameterInit:
//-----------------------------------------------------------------------------
//
//  HAUD 2024.07.04
//
// 
//  - hard coded station parameter
//-----------------------------------------------------------------------------
//-----------------------------------------------------------------------------

//-----------------------------------------------------------------------------------------------------------------------------------------
//  LOAD
    sStationText  := 'LOAD 1/5';
//-----------------------------------------------------------------------------------------------------------------------------------------
nStationParameter := 1;
GVL_XTS.StationParameter[nStationParameter].sText                 := 'LOAD 1/5';
GVL_XTS.StationParameter[nStationParameter].rPosWait              :=     20.0;  // absolute modulo position

GVL_XTS.StationParameter[nStationParameter].nConfiguredStopCount  :=      1;   // how many stops the mover has to make in this station
GVL_XTS.StationParameter[nStationParameter].rPosStop[1]           :=    100.0; // relative to rPosWait

GVL_XTS.StationParameter[nStationParameter].rReleaseDistance      :=    500.0; // relative to Mover.ActPos

GVL_XTS.StationParameter[nStationParameter].rGap                  :=     95.0;
GVL_XTS.StationParameter[nStationParameter].rVelo                 :=   2500.0;
GVL_XTS.StationParameter[nStationParameter].rAccDec               :=  15000.0;
GVL_XTS.StationParameter[nStationParameter].rJerk                 := 800000.0;

//-----------------------------------------------------------------------------------------------------------------------------------------
nStationParameter := 2;
GVL_XTS.StationParameter[nStationParameter].sText                 := 'LOAD 2/5';
GVL_XTS.StationParameter[nStationParameter].rPosWait              :=     20.0;  // absolute modulo position

GVL_XTS.StationParameter[nStationParameter].nConfiguredStopCount  :=      1;   // how many stops the mover has to make in this station
GVL_XTS.StationParameter[nStationParameter].rPosStop[1]           :=    200.0; // relative to rPosWait

GVL_XTS.StationParameter[nStationParameter].rReleaseDistance      :=    400.0; // relative to Mover.ActPos

GVL_XTS.StationParameter[nStationParameter].rGap                  :=     95.0;
GVL_XTS.StationParameter[nStationParameter].rVelo                 :=   2500.0;
GVL_XTS.StationParameter[nStationParameter].rAccDec               :=  15000.0;
GVL_XTS.StationParameter[nStationParameter].rJerk                 := 800000.0;

//-----------------------------------------------------------------------------------------------------------------------------------------
nStationParameter := 3;
GVL_XTS.StationParameter[nStationParameter].sText                 := 'LOAD 3/5';
GVL_XTS.StationParameter[nStationParameter].rPosWait              :=     20.0;  // absolute modulo position

GVL_XTS.StationParameter[nStationParameter].nConfiguredStopCount  :=      1;   // how many stops the mover has to make in this station
GVL_XTS.StationParameter[nStationParameter].rPosStop[1]           :=    300.0; // relative to rPosWait

GVL_XTS.StationParameter[nStationParameter].rReleaseDistance      :=    300.0; // relative to Mover.ActPos

GVL_XTS.StationParameter[nStationParameter].rGap                  :=     95.0;
GVL_XTS.StationParameter[nStationParameter].rVelo                 :=   2500.0;
GVL_XTS.StationParameter[nStationParameter].rAccDec               :=  15000.0;
GVL_XTS.StationParameter[nStationParameter].rJerk                 := 800000.0;

//-----------------------------------------------------------------------------------------------------------------------------------------
nStationParameter := 4;
GVL_XTS.StationParameter[nStationParameter].sText                 := 'LOAD 4/5';
GVL_XTS.StationParameter[nStationParameter].rPosWait              :=     20.0;  // absolute modulo position

GVL_XTS.StationParameter[nStationParameter].nConfiguredStopCount  :=      1;   // how many stops the mover has to make in this station
GVL_XTS.StationParameter[nStationParameter].rPosStop[1]           :=    400.0; // relative to rPosWait

GVL_XTS.StationParameter[nStationParameter].rReleaseDistance      :=    200.0; // relative to Mover.ActPos

GVL_XTS.StationParameter[nStationParameter].rGap                  :=     95.0;
GVL_XTS.StationParameter[nStationParameter].rVelo                 :=   1250.0;
GVL_XTS.StationParameter[nStationParameter].rAccDec               :=  15000.0;
GVL_XTS.StationParameter[nStationParameter].rJerk                 := 800000.0;

//-----------------------------------------------------------------------------------------------------------------------------------------
nStationParameter := 5;
GVL_XTS.StationParameter[nStationParameter].sText                 := 'LOAD 5/5';
GVL_XTS.StationParameter[nStationParameter].rPosWait              :=     20.0;  // absolute modulo position

GVL_XTS.StationParameter[nStationParameter].nConfiguredStopCount  :=      1;   // how many stops the mover has to make in this station
GVL_XTS.StationParameter[nStationParameter].rPosStop[1]           :=    500.0; // relative to rPosWait

GVL_XTS.StationParameter[nStationParameter].rReleaseDistance      :=    150.0; // relative to Mover.ActPos

GVL_XTS.StationParameter[nStationParameter].rGap                  :=     95.0;
GVL_XTS.StationParameter[nStationParameter].rVelo                 :=   1250.0;
GVL_XTS.StationParameter[nStationParameter].rAccDec               :=  15000.0;
GVL_XTS.StationParameter[nStationParameter].rJerk                 := 800000.0;

//-----------------------------------------------------------------------------------------------------------------------------------------
//-----------------------------------------------------------------------------------------------------------------------------------------
//  WKZ_1
    sStationText  := 'WORK_1 1/5';
//-----------------------------------------------------------------------------------------------------------------------------------------
//-----------------------------------------------------------------------------------------------------------------------------------------
nStationParameter := 6;
GVL_XTS.StationParameter[nStationParameter].sText                 := 'WORK_1 1/5';
GVL_XTS.StationParameter[nStationParameter].rPosWait              :=   1820.0;  // absolute modulo position

GVL_XTS.StationParameter[nStationParameter].nConfiguredStopCount  :=      1;   // how many stops the mover has to make in this station
GVL_XTS.StationParameter[nStationParameter].rPosStop[1]           :=    100.0; // relative to rPosWait

GVL_XTS.StationParameter[nStationParameter].rReleaseDistance      :=    500.0; // relative to Mover.ActPos

GVL_XTS.StationParameter[nStationParameter].rGap                  :=     95.0;
GVL_XTS.StationParameter[nStationParameter].rVelo                 :=   2500.0;
GVL_XTS.StationParameter[nStationParameter].rAccDec               :=  15000.0;
GVL_XTS.StationParameter[nStationParameter].rJerk                 := 800000.0;

//-----------------------------------------------------------------------------------------------------------------------------------------
nStationParameter := 7;
GVL_XTS.StationParameter[nStationParameter].sText                 := 'WORK_1 2/5';
GVL_XTS.StationParameter[nStationParameter].rPosWait              :=   1820.0;  // absolute modulo position

GVL_XTS.StationParameter[nStationParameter].nConfiguredStopCount  :=      1;   // how many stops the mover has to make in this station
GVL_XTS.StationParameter[nStationParameter].rPosStop[1]           :=    200.0; // relative to rPosWait

GVL_XTS.StationParameter[nStationParameter].rReleaseDistance      :=    400.0; // relative to Mover.ActPos

GVL_XTS.StationParameter[nStationParameter].rGap                  :=     95.0;
GVL_XTS.StationParameter[nStationParameter].rVelo                 :=   2500.0;
GVL_XTS.StationParameter[nStationParameter].rAccDec               :=  15000.0;
GVL_XTS.StationParameter[nStationParameter].rJerk                 := 800000.0;

//-----------------------------------------------------------------------------------------------------------------------------------------
nStationParameter := 8;
GVL_XTS.StationParameter[nStationParameter].sText                 := 'WORK_1 3/5';
GVL_XTS.StationParameter[nStationParameter].rPosWait              :=   1820.0;  // absolute modulo position

GVL_XTS.StationParameter[nStationParameter].nConfiguredStopCount  :=      1;   // how many stops the mover has to make in this station
GVL_XTS.StationParameter[nStationParameter].rPosStop[1]           :=    300.0; // relative to rPosWait

GVL_XTS.StationParameter[nStationParameter].rReleaseDistance      :=    300.0; // relative to Mover.ActPos

GVL_XTS.StationParameter[nStationParameter].rGap                  :=     95.0;
GVL_XTS.StationParameter[nStationParameter].rVelo                 :=   2500.0;
GVL_XTS.StationParameter[nStationParameter].rAccDec               :=  15000.0;
GVL_XTS.StationParameter[nStationParameter].rJerk                 := 800000.0;

//-----------------------------------------------------------------------------------------------------------------------------------------
nStationParameter := 9;
GVL_XTS.StationParameter[nStationParameter].sText                 := 'WORK_1 4/5';
GVL_XTS.StationParameter[nStationParameter].rPosWait              :=   1820.0;  // absolute modulo position

GVL_XTS.StationParameter[nStationParameter].nConfiguredStopCount  :=      1;   // how many stops the mover has to make in this station
GVL_XTS.StationParameter[nStationParameter].rPosStop[1]           :=    400.0; // relative to rPosWait

GVL_XTS.StationParameter[nStationParameter].rReleaseDistance      :=    200.0; // relative to Mover.ActPos

GVL_XTS.StationParameter[nStationParameter].rGap                  :=     95.0;
GVL_XTS.StationParameter[nStationParameter].rVelo                 :=   1250.0;
GVL_XTS.StationParameter[nStationParameter].rAccDec               :=  15000.0;
GVL_XTS.StationParameter[nStationParameter].rJerk                 := 800000.0;

//-----------------------------------------------------------------------------------------------------------------------------------------
nStationParameter := 10;
GVL_XTS.StationParameter[nStationParameter].sText                 := 'WORK_1 5/5';
GVL_XTS.StationParameter[nStationParameter].rPosWait              :=   1820.0;  // absolute modulo position

GVL_XTS.StationParameter[nStationParameter].nConfiguredStopCount  :=      1;   // how many stops the mover has to make in this station
GVL_XTS.StationParameter[nStationParameter].rPosStop[1]           :=    500.0; // relative to rPosWait

GVL_XTS.StationParameter[nStationParameter].rReleaseDistance      :=    150.0; // relative to Mover.ActPos

GVL_XTS.StationParameter[nStationParameter].rGap                  :=     95.0;
GVL_XTS.StationParameter[nStationParameter].rVelo                 :=   1250.0;
GVL_XTS.StationParameter[nStationParameter].rAccDec               :=  15000.0;
GVL_XTS.StationParameter[nStationParameter].rJerk                 := 800000.0;

//-----------------------------------------------------------------------------------------------------------------------------------------
//-----------------------------------------------------------------------------------------------------------------------------------------
//  DISTRIBUTOR_SCAN
    sStationText  := 'DISTRIBUTOR_SCAN';
//-----------------------------------------------------------------------------------------------------------------------------------------
//-----------------------------------------------------------------------------------------------------------------------------------------
nStationParameter := 11;
GVL_XTS.StationParameter[nStationParameter].sText                 := 'DISTRIBUTOR_SCAN';
GVL_XTS.StationParameter[nStationParameter].rPosWait              :=   2750.0;  // absolute modulo position

GVL_XTS.StationParameter[nStationParameter].nConfiguredStopCount  :=      1;   // how many stops the mover has to make in this station
GVL_XTS.StationParameter[nStationParameter].rPosStop[1]           :=      0.0; // relative to rPosWait

GVL_XTS.StationParameter[nStationParameter].rReleaseDistance      :=    -10.0; // relative to Mover.ActPos

GVL_XTS.StationParameter[nStationParameter].rGap                  :=     95.0;
GVL_XTS.StationParameter[nStationParameter].rVelo                 :=   3000.0;
GVL_XTS.StationParameter[nStationParameter].rAccDec               :=  15000.0;
GVL_XTS.StationParameter[nStationParameter].rJerk                 := 800000.0;


//-----------------------------------------------------------------------------------------------------------------------------------------
//-----------------------------------------------------------------------------------------------------------------------------------------
//  SCANNER_1
    sStationText  := 'SCANNER 1/2';
//-----------------------------------------------------------------------------------------------------------------------------------------
//-----------------------------------------------------------------------------------------------------------------------------------------
nStationParameter := 12;
GVL_XTS.StationParameter[nStationParameter].sText                 := 'SCANNER 1/2';
GVL_XTS.StationParameter[nStationParameter].rPosWait              :=   3400.0;  // absolute modulo position

GVL_XTS.StationParameter[nStationParameter].nConfiguredStopCount  :=      1;   // how many stops the mover has to make in this station
GVL_XTS.StationParameter[nStationParameter].rPosStop[1]           :=    100.0; // relative to rPosWait

GVL_XTS.StationParameter[nStationParameter].rReleaseDistance      :=     20.0; // relative to Mover.ActPos

GVL_XTS.StationParameter[nStationParameter].rGap                  :=     95.0;
GVL_XTS.StationParameter[nStationParameter].rVelo                 :=   3000.0;
GVL_XTS.StationParameter[nStationParameter].rAccDec               :=  15000.0;
GVL_XTS.StationParameter[nStationParameter].rJerk                 := 800000.0;

//-----------------------------------------------------------------------------------------------------------------------------------------
//-----------------------------------------------------------------------------------------------------------------------------------------
//  SCANNER_2
    sStationText  := 'SCANNER 2/2';
//-----------------------------------------------------------------------------------------------------------------------------------------
//-----------------------------------------------------------------------------------------------------------------------------------------
nStationParameter := 13;
GVL_XTS.StationParameter[nStationParameter].sText                 := 'SCANNER 2/2';
GVL_XTS.StationParameter[nStationParameter].rPosWait              :=   3400.0;  // absolute modulo position

GVL_XTS.StationParameter[nStationParameter].nConfiguredStopCount  :=      1;   // how many stops the mover has to make in this station
GVL_XTS.StationParameter[nStationParameter].rPosStop[1]           :=    200.0; // relative to rPosWait

GVL_XTS.StationParameter[nStationParameter].rReleaseDistance      :=     10.0; // relative to Mover.ActPos

GVL_XTS.StationParameter[nStationParameter].rGap                  :=     95.0;
GVL_XTS.StationParameter[nStationParameter].rVelo                 :=   3000.0;
GVL_XTS.StationParameter[nStationParameter].rAccDec               :=  15000.0;
GVL_XTS.StationParameter[nStationParameter].rJerk                 := 800000.0;

//-----------------------------------------------------------------------------------------------------------------------------------------
//-----------------------------------------------------------------------------------------------------------------------------------------
//  DISTRIBUTOR_WKZ2
    sStationText  := 'DISTRIBUTOR_WORK_2';
//-----------------------------------------------------------------------------------------------------------------------------------------
//-----------------------------------------------------------------------------------------------------------------------------------------
nStationParameter := 14;
GVL_XTS.StationParameter[nStationParameter].sText                 := 'DISTRIBUTOR_WORK_2';
GVL_XTS.StationParameter[nStationParameter].rPosWait              :=   4000.0;  // absolute modulo position

GVL_XTS.StationParameter[nStationParameter].nConfiguredStopCount  :=      1;   // how many stops the mover has to make in this station
GVL_XTS.StationParameter[nStationParameter].rPosStop[1]           :=      0.0; // relative to rPosWait

GVL_XTS.StationParameter[nStationParameter].rReleaseDistance      :=    -10.0; // relative to Mover.ActPos

GVL_XTS.StationParameter[nStationParameter].rGap                  :=     95.0;
GVL_XTS.StationParameter[nStationParameter].rVelo                 :=   1250.0;
GVL_XTS.StationParameter[nStationParameter].rAccDec               :=  15000.0;
GVL_XTS.StationParameter[nStationParameter].rJerk                 := 800000.0;

//-----------------------------------------------------------------------------------------------------------------------------------------
//-----------------------------------------------------------------------------------------------------------------------------------------
//  WKZ_2
    sStationText  := 'WORK_2 1/5';
//-----------------------------------------------------------------------------------------------------------------------------------------
//-----------------------------------------------------------------------------------------------------------------------------------------
nStationParameter := 15;
GVL_XTS.StationParameter[nStationParameter].sText                 := 'WORK_2 1/5';
GVL_XTS.StationParameter[nStationParameter].rPosWait              :=   5300.0;  // absolute modulo position

GVL_XTS.StationParameter[nStationParameter].nConfiguredStopCount  :=      1;   // how many stops the mover has to make in this station
GVL_XTS.StationParameter[nStationParameter].rPosStop[1]           :=    100.0; // relative to rPosWait

GVL_XTS.StationParameter[nStationParameter].rReleaseDistance      :=    200.0; // relative to Mover.ActPos

GVL_XTS.StationParameter[nStationParameter].rGap                  :=     95.0;
GVL_XTS.StationParameter[nStationParameter].rVelo                 :=   2500.0;
GVL_XTS.StationParameter[nStationParameter].rAccDec               :=  15000.0;
GVL_XTS.StationParameter[nStationParameter].rJerk                 := 800000.0;

//-----------------------------------------------------------------------------------------------------------------------------------------
nStationParameter := 16;
GVL_XTS.StationParameter[nStationParameter].sText                 := 'WORK_2 2/5';
GVL_XTS.StationParameter[nStationParameter].rPosWait              :=   5300.0;  // absolute modulo position

GVL_XTS.StationParameter[nStationParameter].nConfiguredStopCount  :=      1;   // how many stops the mover has to make in this station
GVL_XTS.StationParameter[nStationParameter].rPosStop[1]           :=    200.0; // relative to rPosWait

GVL_XTS.StationParameter[nStationParameter].rReleaseDistance      :=    150.0; // relative to Mover.ActPos

GVL_XTS.StationParameter[nStationParameter].rGap                  :=     95.0;
GVL_XTS.StationParameter[nStationParameter].rVelo                 :=   2500.0;
GVL_XTS.StationParameter[nStationParameter].rAccDec               :=  15000.0;
GVL_XTS.StationParameter[nStationParameter].rJerk                 := 800000.0;

//-----------------------------------------------------------------------------------------------------------------------------------------
nStationParameter := 17;
GVL_XTS.StationParameter[nStationParameter].sText                 := 'WORK_2 3/5';
GVL_XTS.StationParameter[nStationParameter].rPosWait              :=   5300.0;  // absolute modulo position

GVL_XTS.StationParameter[nStationParameter].nConfiguredStopCount  :=      1;   // how many stops the mover has to make in this station
GVL_XTS.StationParameter[nStationParameter].rPosStop[1]           :=    300.0; // relative to rPosWait

GVL_XTS.StationParameter[nStationParameter].rReleaseDistance      :=    100.0; // relative to Mover.ActPos

GVL_XTS.StationParameter[nStationParameter].rGap                  :=     95.0;
GVL_XTS.StationParameter[nStationParameter].rVelo                 :=   2500.0;
GVL_XTS.StationParameter[nStationParameter].rAccDec               :=  15000.0;
GVL_XTS.StationParameter[nStationParameter].rJerk                 := 800000.0;

//-----------------------------------------------------------------------------------------------------------------------------------------
nStationParameter := 18;
GVL_XTS.StationParameter[nStationParameter].sText                 := 'WORK_2 4/5';
GVL_XTS.StationParameter[nStationParameter].rPosWait              :=   5300.0;  // absolute modulo position

GVL_XTS.StationParameter[nStationParameter].nConfiguredStopCount  :=      1;   // how many stops the mover has to make in this station
GVL_XTS.StationParameter[nStationParameter].rPosStop[1]           :=    400.0; // relative to rPosWait

GVL_XTS.StationParameter[nStationParameter].rReleaseDistance      :=    50.0; // relative to Mover.ActPos

GVL_XTS.StationParameter[nStationParameter].rGap                  :=     95.0;
GVL_XTS.StationParameter[nStationParameter].rVelo                 :=   2500.0;
GVL_XTS.StationParameter[nStationParameter].rAccDec               :=  15000.0;
GVL_XTS.StationParameter[nStationParameter].rJerk                 := 800000.0;

//-----------------------------------------------------------------------------------------------------------------------------------------
nStationParameter := 19;
GVL_XTS.StationParameter[nStationParameter].sText                 := 'WORK_2 5/5';
GVL_XTS.StationParameter[nStationParameter].rPosWait              :=   5300.0;  // absolute modulo position

GVL_XTS.StationParameter[nStationParameter].nConfiguredStopCount  :=      1;   // how many stops the mover has to make in this station
GVL_XTS.StationParameter[nStationParameter].rPosStop[1]           :=    500.0; // relative to rPosWait

GVL_XTS.StationParameter[nStationParameter].rReleaseDistance      :=     10.0; // relative to Mover.ActPos

GVL_XTS.StationParameter[nStationParameter].rGap                  :=     95.0;
GVL_XTS.StationParameter[nStationParameter].rVelo                 :=   1250.0;
GVL_XTS.StationParameter[nStationParameter].rAccDec               :=  15000.0;
GVL_XTS.StationParameter[nStationParameter].rJerk                 := 800000.0;

//-----------------------------------------------------------------------------------------------------------------------------------------
//-----------------------------------------------------------------------------------------------------------------------------------------
//  CAMERA_ADJUST
    sStationText  := 'INSPECT';
//-----------------------------------------------------------------------------------------------------------------------------------------
//-----------------------------------------------------------------------------------------------------------------------------------------
nStationParameter := 20;
GVL_XTS.StationParameter[nStationParameter].sText                 := 'INSPECT';
GVL_XTS.StationParameter[nStationParameter].rPosWait              :=   6400.0;  // absolute modulo position

GVL_XTS.StationParameter[nStationParameter].nConfiguredStopCount  :=      1;   // how many stops the mover has to make in this station
GVL_XTS.StationParameter[nStationParameter].rPosStop[1]           :=    100.0; // relative to rPosWait

GVL_XTS.StationParameter[nStationParameter].rReleaseDistance      :=     5.0; // relative to Mover.ActPos

GVL_XTS.StationParameter[nStationParameter].rGap                  :=     95.0;
GVL_XTS.StationParameter[nStationParameter].rVelo                 :=   2500.0;
GVL_XTS.StationParameter[nStationParameter].rAccDec               :=  17500.0;
GVL_XTS.StationParameter[nStationParameter].rJerk                 := 800000.0;

//-----------------------------------------------------------------------------------------------------------------------------------------
//-----------------------------------------------------------------------------------------------------------------------------------------
//  DISTRIBUTOR_CAMERA
    sStationText  := 'DISTRIBUTOR_CAMERA';
//-----------------------------------------------------------------------------------------------------------------------------------------
//-----------------------------------------------------------------------------------------------------------------------------------------
nStationParameter := 21;
GVL_XTS.StationParameter[nStationParameter].sText                 := 'DISTRIBUTOR_CAMERA';
GVL_XTS.StationParameter[nStationParameter].rPosWait              :=   6600.0;  // absolute modulo position

GVL_XTS.StationParameter[nStationParameter].nConfiguredStopCount  :=      1;   // how many stops the mover has to make in this station
GVL_XTS.StationParameter[nStationParameter].rPosStop[1]           :=      0.0; // relative to rPosWait

GVL_XTS.StationParameter[nStationParameter].rReleaseDistance      :=    -10.0; // relative to Mover.ActPos

GVL_XTS.StationParameter[nStationParameter].rGap                  :=     95.0;
GVL_XTS.StationParameter[nStationParameter].rVelo                 :=   2500.0;
GVL_XTS.StationParameter[nStationParameter].rAccDec               :=  17500.0;
GVL_XTS.StationParameter[nStationParameter].rJerk                 := 800000.0;

//-----------------------------------------------------------------------------------------------------------------------------------------
//-----------------------------------------------------------------------------------------------------------------------------------------
//  CAMERA
    sStationText  := 'CAMERA 1/3';
//-----------------------------------------------------------------------------------------------------------------------------------------
//-----------------------------------------------------------------------------------------------------------------------------------------
nStationParameter := 22;
GVL_XTS.StationParameter[nStationParameter].sText                 := 'CAMERA 1/3';
GVL_XTS.StationParameter[nStationParameter].rPosWait              :=   7000.0;  // absolute modulo position

GVL_XTS.StationParameter[nStationParameter].nConfiguredStopCount  :=      1;   // how many stops the mover has to make in this station
GVL_XTS.StationParameter[nStationParameter].rPosStop[1]           :=    200.0; // relative to rPosWait

GVL_XTS.StationParameter[nStationParameter].rReleaseDistance      :=    100.0; // relative to Mover.ActPos

GVL_XTS.StationParameter[nStationParameter].rGap                  :=     95.0;
GVL_XTS.StationParameter[nStationParameter].rVelo                 :=   1250.0;
GVL_XTS.StationParameter[nStationParameter].rAccDec               :=  15000.0;
GVL_XTS.StationParameter[nStationParameter].rJerk                 := 800000.0;

//-----------------------------------------------------------------------------------------------------------------------------------------
nStationParameter := 23;
GVL_XTS.StationParameter[nStationParameter].sText                 := 'CAMERA 2/3';
GVL_XTS.StationParameter[nStationParameter].rPosWait              :=   7000.0;  // absolute modulo position

GVL_XTS.StationParameter[nStationParameter].nConfiguredStopCount  :=      1;   // how many stops the mover has to make in this station
GVL_XTS.StationParameter[nStationParameter].rPosStop[1]           :=    400.0; // relative to rPosWait

GVL_XTS.StationParameter[nStationParameter].rReleaseDistance      :=    50.0; // relative to Mover.ActPos

GVL_XTS.StationParameter[nStationParameter].rGap                  :=     95.0;
GVL_XTS.StationParameter[nStationParameter].rVelo                 :=   1250.0;
GVL_XTS.StationParameter[nStationParameter].rAccDec               :=  15000.0;
GVL_XTS.StationParameter[nStationParameter].rJerk                 := 800000.0;

//-----------------------------------------------------------------------------------------------------------------------------------------
nStationParameter := 24;
GVL_XTS.StationParameter[nStationParameter].sText                 := 'CAMERA 3/3';
GVL_XTS.StationParameter[nStationParameter].rPosWait              :=   7000.0;  // absolute modulo position

GVL_XTS.StationParameter[nStationParameter].nConfiguredStopCount  :=      1;   // how many stops the mover has to make in this station
GVL_XTS.StationParameter[nStationParameter].rPosStop[1]           :=    600.0; // relative to rPosWait

GVL_XTS.StationParameter[nStationParameter].rReleaseDistance      :=     10.0; // relative to Mover.ActPos

GVL_XTS.StationParameter[nStationParameter].rGap                  :=     95.0;
GVL_XTS.StationParameter[nStationParameter].rVelo                 :=   1250.0;
GVL_XTS.StationParameter[nStationParameter].rAccDec               :=  15000.0;
GVL_XTS.StationParameter[nStationParameter].rJerk                 := 800000.0;

//-----------------------------------------------------------------------------------------------------------------------------------------
//-----------------------------------------------------------------------------------------------------------------------------------------
//  DISTRIBUTOR_UNLOAD
    sStationText  := 'DISTRIBUTOR_UNLOAD';
//-----------------------------------------------------------------------------------------------------------------------------------------
//-----------------------------------------------------------------------------------------------------------------------------------------
nStationParameter := 25;
GVL_XTS.StationParameter[nStationParameter].sText                 := 'DISTRIBUTOR_UNLOAD';
GVL_XTS.StationParameter[nStationParameter].rPosWait              :=   9000.0;  // absolute modulo position

GVL_XTS.StationParameter[nStationParameter].nConfiguredStopCount  :=      1;   // how many stops the mover has to make in this station
GVL_XTS.StationParameter[nStationParameter].rPosStop[1]           :=      0.0; // relative to rPosWait

GVL_XTS.StationParameter[nStationParameter].rReleaseDistance      :=    100.0; // relative to Mover.ActPos

GVL_XTS.StationParameter[nStationParameter].rGap                  :=     95.0;
GVL_XTS.StationParameter[nStationParameter].rVelo                 :=   1250.0;
GVL_XTS.StationParameter[nStationParameter].rAccDec               :=  15000.0;
GVL_XTS.StationParameter[nStationParameter].rJerk                 := 800000.0;

//-----------------------------------------------------------------------------------------------------------------------------------------
//-----------------------------------------------------------------------------------------------------------------------------------------
//  UNLOAD
    sStationText  := 'UNLOAD 1/2';
//-----------------------------------------------------------------------------------------------------------------------------------------
//-----------------------------------------------------------------------------------------------------------------------------------------
nStationParameter := 26;
GVL_XTS.StationParameter[nStationParameter].sText                 := 'UNLOAD 1/2';
GVL_XTS.StationParameter[nStationParameter].rPosWait              :=  10000.0;  // absolute modulo position

GVL_XTS.StationParameter[nStationParameter].nConfiguredStopCount  :=      1;   // how many stops the mover has to make in this station
GVL_XTS.StationParameter[nStationParameter].rPosStop[1]           :=    100.0; // relative to rPosWait

GVL_XTS.StationParameter[nStationParameter].rReleaseDistance      :=    400.0; // relative to Mover.ActPos

GVL_XTS.StationParameter[nStationParameter].rGap                  :=     95.0;
GVL_XTS.StationParameter[nStationParameter].rVelo                 :=   2500.0;
GVL_XTS.StationParameter[nStationParameter].rAccDec               :=  15000.0;
GVL_XTS.StationParameter[nStationParameter].rJerk                 := 800000.0;

//-----------------------------------------------------------------------------------------------------------------------------------------
nStationParameter := 27;
GVL_XTS.StationParameter[nStationParameter].sText                 := 'UNLOAD 1/2';
GVL_XTS.StationParameter[nStationParameter].rPosWait              :=  10000.0;  // absolute modulo position

GVL_XTS.StationParameter[nStationParameter].nConfiguredStopCount  :=      1;   // how many stops the mover has to make in this station
GVL_XTS.StationParameter[nStationParameter].rPosStop[1]           :=    200.0; // relative to rPosWait

GVL_XTS.StationParameter[nStationParameter].rReleaseDistance      :=    200.0; // relative to Mover.ActPos

GVL_XTS.StationParameter[nStationParameter].rGap                  :=     95.0;
GVL_XTS.StationParameter[nStationParameter].rVelo                 :=   2500.0;
GVL_XTS.StationParameter[nStationParameter].rAccDec               :=  15000.0;
GVL_XTS.StationParameter[nStationParameter].rJerk                 := 800000.0;

//-----------------------------------------------------------------------------------------------------------------------------------------
//-----------------------------------------------------------------------------------------------------------------------------------------
//  DISTRIBUTOR_LOAD
    sStationText  := 'DISTRIBUTOR_LOAD';
//-----------------------------------------------------------------------------------------------------------------------------------------
//-----------------------------------------------------------------------------------------------------------------------------------------
nStationParameter := 28;
GVL_XTS.StationParameter[nStationParameter].sText                 := 'DISTRIBUTOR_LOAD';
GVL_XTS.StationParameter[nStationParameter].rPosWait              :=  11000.0;  // absolute modulo position

GVL_XTS.StationParameter[nStationParameter].nConfiguredStopCount  :=      1;   // how many stops the mover has to make in this station
GVL_XTS.StationParameter[nStationParameter].rPosStop[1]           :=      0.0; // relative to rPosWait

GVL_XTS.StationParameter[nStationParameter].rReleaseDistance      :=    -10.0; // relative to Mover.ActPos

GVL_XTS.StationParameter[nStationParameter].rGap                  :=     95.0;
GVL_XTS.StationParameter[nStationParameter].rVelo                 :=   1500.0;
GVL_XTS.StationParameter[nStationParameter].rAccDec               :=  15000.0;
GVL_XTS.StationParameter[nStationParameter].rJerk                 := 800000.0;
END_ACTION

METHOD VisuData
VAR_INPUT
END_VAR

// get enumerations from XPU for visu:
eTransportState                       := f_GetState   (GVL_XTS.XtsTransportState.State);
eTransportResult                      := f_GetProgress(GVL_XTS.XtsTransportState.State);

eXpuState                             := f_GetState   (GVL_XTS.XtsTransportState.XpuState.State);
eXpuResult                            := f_GetProgress(GVL_XTS.XtsTransportState.XpuState.State);

eXpuCheck                             := GVL_XTS.XtsTransportState.XpuState.Check;

// display xpu state and result in visu
// get strings and info
sCaGroupState                         := TO_STRING(GVL_XTS.XtsTransportState.GroupInfo.CaGroupState);

sTransportState                       := TO_STRING(eTransportState);
sTransportCheck                       := TO_STRING(GVL_XTS.XtsTransportState.Check);
sTransportResult                      := TO_STRING(eTransportResult);

sXpuState                             := TO_STRING(eXpuState);
sXpuResult                            := TO_STRING(eXpuResult);
sXpuCheck                             := TO_STRING(eXpuCheck);

sXpuOpMode                            := f_XpuOperationModeToString         (GVL_XTS.XtsTransportState.XpuInfo.OperationMode);
sXpuMoverdetectionMode                := f_MoverIdDetectionModeToString     (GVL_XTS.XtsTransportState.XpuInfo.IdDetectionMode);
sXpuMoverAssignement                  := f_MoverPositionAssignementToString (GVL_XTS.XtsTransportState.XpuInfo.MoverPositionAssignement);

nMoverSelected                        := SEL((nMoverSelected<1), nMoverSelected, 1);
nMoverSelected                        := SEL((nMoverSelected>MAX_MOVER), nMoverSelected, MAX_MOVER);

nStationSelected                      := SEL((nStationSelected<1), nStationSelected, 1);
nStationSelected                      := SEL((nStationSelected>MAX_STATION), nStationSelected, MAX_STATION);

nProcessSelected                      := SEL((nProcessSelected<1), nProcessSelected, 1);
nProcessSelected                      := SEL((nProcessSelected>MAX_PROCESS), nProcessSelected, MAX_PROCESS);

bStationEnable                        := SEL((GVL_XTS.StationCtrl[nStationSelected].eCmd = E_STATION_CTRL.STATION_ENABLE),        FALSE, TRUE);
bStationEnter                         := SEL((GVL_XTS.StationCtrl[nStationSelected].eCmd = E_STATION_CTRL.STATION_MOVER_ENTER),   FALSE, TRUE);
bStationStart                         := SEL((GVL_XTS.StationCtrl[nStationSelected].eCmd = E_STATION_CTRL.STATION_PROCESS_START), FALSE, TRUE);
bStationDone                          := SEL((GVL_XTS.StationCtrl[nStationSelected].eCmd = E_STATION_CTRL.STATION_PROCESS_DONE),  FALSE, TRUE);
bStationOut                           := SEL((GVL_XTS.StationCtrl[nStationSelected].eCmd = E_STATION_CTRL.STATION_MOVER_OUT),     FALSE, TRUE);
bStationGone                          := SEL((GVL_XTS.StationCtrl[nStationSelected].eCmd = E_STATION_CTRL.STATION_MOVER_GONE),    FALSE, TRUE);

sStationState                         := TO_STRING(GVL_XTS.StationState[nStationSelected].eState);
sStationStateMask                     := Tc2_Utilities.BYTE_TO_BINSTR(GVL_XTS.StationState[nStationSelected].nMask, 8);
sStationCtrlMask                      := Tc2_Utilities.BYTE_TO_BINSTR(GVL_XTS.StationCtrl[nStationSelected].nMask, 8);

sProcessEnableMask                    := Tc2_Utilities.DWORD_TO_BINSTR(GVL_PROCESS.Process[nProcessSelected].EnableProcess, 16);
END_METHOD

END_PROGRAM

// ---- XTS/_types/f_MoverIdDetectionModeToString.TcPOU
FUNCTION f_MoverIdDetectionModeToString : string(20)
VAR_INPUT
  nDetectionMode    : UINT;
END_VAR
VAR
END_VAR


CASE nDetectionMode
OF
  0:
    f_MoverIdDetectionModeToString  := 'Standard';
  1:
    f_MoverIdDetectionModeToString  := 'Mover 1';
  2:
    f_MoverIdDetectionModeToString  := 'Multiple Mover 1';
ELSE
    f_MoverIdDetectionModeToString  := 'UNKNOWN Mode';
END_CASE

END_FUNCTION

// ---- XTS/_types/f_MoverPositionAssignementToString.TcPOU
FUNCTION f_MoverPositionAssignementToString : string(30)
VAR_INPUT
  nPosAssignement   : UINT;
END_VAR
VAR
END_VAR


CASE nPosAssignement
OF
  0:
    f_MoverPositionAssignementToString    := 'Standard';
  1:
    f_MoverPositionAssignementToString    := 'Start At First Mover';
ELSE
    f_MoverPositionAssignementToString    := 'UNKNOWN Assignement';
END_CASE

END_FUNCTION

// ---- PROCESS/fb_Process.TcPOU
//---------------------------------------------------------------------------------------------------------------
//
//  HAUD 2023.03.27
//
//  TR08
//  - XTS_TRANSPORT_LAYER
//
//  fb_Process
//  - grouping of xts stations to sync start process
//  - nFirst to nLast xts stations are checked for starting process simultaneously
//  - basic preparation of station target index in PrepareTarget()
//  - handshake with station control for mover transport through station
//
//---------------------------------------------------------------------------------------------------------------
// This SOFTWARE is provided as an Exemple by THE PROVIDER "as is" and "with all faults." THE PROVIDER makes no 
// representations or warranties of any kind concerning the safety, suitability, lack of viruses, inaccuracies, 
// typographical errors, or other harmful components of this SOFTWARE. There are inherent dangers in the use of 
// any software, and you are solely responsible for determining whether this SOFTWARE is compatible with your 
// equipment and other software installed on your equipment. You are also solely responsible for the protection 
// of your equipment and backup of your data, and THE PROVIDER will not be liable for any damages you may suffer 
// in connection with using, modifying, or distributing this SOFTWARE.
//---------------------------------------------------------------------------------------------------------------
FUNCTION_BLOCK fb_Process IMPLEMENTS I_ExternControl_Process
VAR
  _eType                      : E_PROCESS_TYPE;   // types of process: SINGLE, PARALLEL, SERIAL, DISTRIBUTOR
  _sCheck                     : STRING;

  _eProcessCmd                : E_STATION_CTRL;   // control from property
  _eProcessState              : E_STATION_STATE;  // state   to   property

  {attribute 'displaymode':='bin'}
  _wEnableProcess             : DWORD; // control sets bits to switch on stations
  _bEnabledStation            : POINTER TO ARRAY[1..XTS_Parameter.MAX_STATION]  OF BOOL; // information about all enabled xts stations

  // xts stations
  _stCtrl                     : POINTER TO ARRAY[1..XTS_Parameter.MAX_STATION]  OF ST_STATION_CTRL;
  _stState                    : POINTER TO ARRAY[1..XTS_Parameter.MAX_STATION]  OF ST_STATION_STATE;

  // who is included in process
  // _nFirst to _nLast MUST be in closed consecutive order
  _nStation,
  _nStationCount,
  _nFirstStation,
  _nLastStation               : UINT;

  // work vars for writing onto _stCtrl[nStation].nTargetStation
  _nTarget,
  _nFirstTarget,
  _nLastTarget                : UINT;   // for parallel process xts stations and the last xts station in serial process

  _nSerialTarget              : ARRAY[1..XTS_Parameter.MAX_STATION]  OF UINT; // serial targets within process

  _nPreparedTarget            : ARRAY[1..XTS_Parameter.MAX_MOVER]  OF UINT;   // targets for parallel and single process

  // bitmasks for station states in CycleStation()
  {attribute 'displaymode':='bin'}
  _wEnable                    : DWORD;   // commanded enable of xts station
  {attribute 'displaymode':='bin'}
  _wEnter                     : DWORD;   // mover asking for entry into xts station
  {attribute 'displaymode':='bin'}
  _wStart                     : DWORD;   // xts station asking for process handshake
  {attribute 'displaymode':='bin'}
  _wLeave                     : DWORD;   // xts station wants to send out mover
  {attribute 'displaymode':='bin'}
  _wQueue                     : DWORD;   // mover was entered into xts station list
  {attribute 'displaymode':='bin'}
  _wMoverInStation            : DWORD;   // mover entry was granted, mover is now in station
  {attribute 'displaymode':='bin'}
  _wError                     : DWORD;   // minor error, must be fixed by _stCtrl[nStation]
  {attribute 'displaymode':='bin'}
  _wErrorFatal                : DWORD;   // fatal error, must be fixed by debugging
  {attribute 'displaymode':='bin'}
  _wTargetId                  : DWORD;   // nTargetStation > 0 in _stDtrl[nStation].nTargetStation

  {attribute 'displaymode':='bin'}
  _TargetMask                 : DWORD;   // bit positions correspond to index of xts station
 
  _bNext                      : BOOL;

  _nProcessPerMinute          : uint; // sum of all xts stations output per minute in process
  _rtrigProcess               : ARRAY[1..XTS_Parameter.MAX_STATION] OF Tc2_Standard.R_TRIG;
  _tonPartsPerMinute          : Tc2_Standard.TON;

  _nMoverPerMinute            : POINTER TO ARRAY[1..XTS_Parameter.MAX_STATION]  OF UINT;
  _nMoverCount,
  _nMoverCountOld             : ARRAY[1..XTS_Parameter.MAX_STATION]  OF UINT;

  _eDistributorTarget         : E_PROGRESS;

END_VAR

METHOD private Check : BOOL

IF (_nFirstStation < 1) OR
   (_nFirstStation > MAX_STATION)
THEN
  _sCheck                     := '_nFirstStation out of bounds';
  RETURN;
END_IF

IF (_nLastStation < 1) OR
   (_nLastStation > MAX_STATION)
THEN
  _sCheck                     := '_nLastStation out of bounds';
  RETURN;
END_IF

IF (_nFirstTarget < 1) OR
   (_nFirstTarget > MAX_STATION)
THEN
  _sCheck                     := '_nFirstTarget out of bounds';
  RETURN;
END_IF

IF (_nLastTarget < 1) OR
   (_nLastTarget > MAX_STATION)
THEN
  _sCheck                     := '_nLastTarget out of bounds';
  RETURN;
END_IF

IF NOT (_stCtrl  <> 0)
THEN
  _sCheck                     := '_stCtrl: missing pointer';
  RETURN;
END_IF

IF NOT (_stState <> 0)
THEN
  _sCheck                     := '_stState: missing pointer';
  RETURN;
END_IF

IF NOT (_bEnabledStation  <> 0)
THEN
  _sCheck                     := '_bEnableStation: missing pointer';
  RETURN;
END_IF

IF not (_nMoverPerMinute <> 0)
THEN
  _sCheck                     := '_nMoverPerMinute: missing pointer';
  RETURN;
END_IF

_nStationCount                := _nLastStation - _nFirstStation + 1;

IF (_nStationCount < 1) OR
   (_nStationCount > (SIZEOF(WORD)*8))
THEN
  _sCheck                     := '_nStationCount out of bounds';
  RETURN;
END_IF


_sCheck                       := TO_STRING(E_PROGRESS.PROGRESS_DONE);
Check                         := TRUE;
END_METHOD

METHOD Cycle
VAR_INST
  _nStn     : uint;
END_VAR
IF NOT Check() THEN RETURN; END_IF


//-----------------------------------------------------------------------------
// collect state information from xts stations
// state information is collected in Masks (WORD), 
// every bit represents one XTS station in process
//-----------------------------------------------------------------------------
//  _wEnable                        : enable cmd was given to xts station
//  _wEnter                         : a mover is requesting entry
//  _wStart                         : mover has arrived and xts station is ready
//  _wLeave                         : xts station wants to send mover out
//  _wQueue                         : somebody's waiting
//  _wMoverInStation                : mover is in station
//  _wError                         : error state for handshake
//  _wErrorFatal                    : error state for severe problems (debugging required)
//  _wTargetId                      : Ctrl.nTargetStation > 0
//  _wMoverInQueueSerial            : SERIAL process: bits to check whether a mover is waiting to be processed
//
CycleStation();                     // get state information from all XtsStations in process
//-----------------------------------------------------------------------------
//-----------------------------------------------------------------------------
//  E_STATION_CTRL.STATION_INIT: hard reset of process and XtsStations
//-----------------------------------------------------------------------------
CASE _eProcessCmd                   // check input property
OF
  E_STATION_CTRL.STATION_INIT:      // commanded init from ctrl
    CASE _eType
    OF
      E_PROCESS_TYPE.SERIAL:
        InitSerialTargets();
    END_CASE
    Init();                         RETURN; // rest you will, return you must
END_CASE
//-----------------------------------------------------------------------------
// E_STATION_STATE.STATION_INIT: pass through here and switch off XtsStations
//-----------------------------------------------------------------------------
CASE _eProcessState                 // check output property
OF
  E_STATION_STATE.STATION_INIT:     // xts station empty, disabled by default
    _eProcessState                  := E_STATION_STATE.STATION_DISABLE;
    FOR _nStn := _nLastStation TO _nFirstStation BY(-1) 
    DO
      _stCtrl^[_nStn].eCmd          := E_STATION_CTRL.STATION_DISABLE;
    END_FOR

END_CASE
//-----------------------------------------------------------------------------
//  E_STATION_STATE.STATION_DISABLE: wait for enable from flow control
//-----------------------------------------------------------------------------
CASE _eProcessState                 // check output property
OF
  E_STATION_STATE.STATION_DISABLE:  // check for enable command
    IF (_eProcessCmd = E_STATION_CTRL.STATION_ENABLE)
    THEN
      _eProcessState                := E_STATION_STATE.STATION_ENABLE;

      FOR _nStn := _nLastStation TO _nFirstStation BY(-1) 
      DO
          _stCtrl^[_nStn].eCmd      := E_STATION_CTRL.STATION_ENABLE;
      END_FOR
    END_IF
END_CASE
//-----------------------------------------------------------------------------
//  E_STATION_STATE.STATION_ENABLE: check Cmd and wait for XtsStations to be enabled
//-----------------------------------------------------------------------------
CASE _eProcessState
OF
  E_STATION_STATE.STATION_ENABLE:
    CASE _eProcessCmd
    OF
      E_STATION_CTRL.STATION_DISABLE:
        _eProcessState              := E_STATION_STATE.STATION_INIT;

